LIN {X 0,Y 261.117,Z 932.425,A -85,B 0,C 180,E1 -18091.542,E2 -18091.542} C_VEL
LIN {X 0,Y 261.103,Z 931.632,A -85,B 0,C 180,E1 -18093.086,E2 -18093.086} C_VEL
LIN {X 0,Y 261.207,Z 929.523,A -85,B 0,C 180,E1 -18095.429,E2 -18095.429} C_VEL
LIN {X 0,Y 261.577,Z 926.266,A -85,B 0,C 180,E1 -18097.72,E2 -18097.72} C_VEL
LIN {X 0,Y 262.252,Z 921.503,A -85,B 0,C 180,E1 -18100.032,E2 -18100.032} C_VEL
LIN {X 0,Y 263.059,Z 916.347,A -85,B 0,C 180,E1 -18101.95,E2 -18101.95} C_VEL
LIN {X 0,Y 263.93,Z 911.311,A -85,B 0,C 180,E1 -18103.474,E2 -18103.474} C_VEL
LIN {X 0,Y 264.941,Z 905.246,A -85,B 0,C 180,E1 -18104.989,E2 -18104.989} C_VEL
LIN {X 0,Y 266.222,Z 897.871,A -85,B 0,C 180,E1 -18106.487,E2 -18106.487} C_VEL
LIN {X 0,Y 267.5,Z 889.973,A -85,B 0,C 180,E1 -18107.784,E2 -18107.784} C_VEL
LIN {X 0,Y 268.675,Z 881.626,A -85,B 0,C 180,E1 -18108.887,E2 -18108.887} C_VEL
LIN {X 0,Y 269.816,Z 871.375,A -85,B 0,C 180,E1 -18109.95,E2 -18109.95} C_VEL
LIN {X 0,Y 270.872,Z 860.075,A -85,B 0,C 180,E1 -18110.756,E2 -18110.756} C_VEL
LIN {X 0,Y 271.49,Z 850.412,A -85,B 0,C 180,E1 -18111.215,E2 -18111.215} C_VEL
LIN {X 0,Y 272.419,Z 812.541,A -85,B 0,C 180,E1 -18112.245,E2 -18112.245} C_VEL
LIN {X 0,Y 268.762,Z 786.761,A -85,B 0,C 180,E1 -18113.292,E2 -18113.292} C_VEL
LIN {X 0,Y 266.245,Z 772.739,A -85,B 0,C 180,E1 -18113.98,E2 -18113.98} C_VEL
LIN {X 0,Y 266.206,Z 769.876,A -85,B 0,C 180,E1 -18114.987,E2 -18114.987} C_VEL
LIN {X 0,Y 264.536,Z 760.93,A -85,B 0,C 180,E1 -18118.751,E2 -18118.751} C_VEL
LIN {X 0,Y 263.188,Z 754.618,A -85,B 0,C 180,E1 -18121.579,E2 -18121.579} C_VEL
LIN {X 0,Y 263.188,Z 754.5,A -85,B 0,C 180,E1 -18125.978,E2 -18125.978} C_VEL
LIN {X 0,Y 263.115,Z 754.506,A -85,B 0,C 180,E1 -18129.871,E2 -18129.871} C_VEL
LIN {X 0,Y 263.124,Z 754.518,A -85,B 0,C 180,E1 -18133.984,E2 -18133.984} C_VEL
LIN {X 0,Y 263.144,Z 754.475,A -85,B 0,C 180,E1 -18138.402,E2 -18138.402} C_VEL
LIN {X 0,Y 263.188,Z 754.456,A -85,B 0,C 180,E1 -18142.108,E2 -18142.108} C_VEL
LIN {X 0,Y 263.184,Z 754.512,A -85,B 0,C 180,E1 -18145.891,E2 -18145.891} C_VEL
LIN {X 0,Y 263.141,Z 754.502,A -85,B 0,C 180,E1 -18149.506,E2 -18149.506} C_VEL
LIN {X 0,Y 263.193,Z 754.509,A -85,B 0,C 180,E1 -18153.003,E2 -18153.003} C_VEL
LIN {X 0,Y 263.186,Z 754.503,A -85,B 0,C 180,E1 -18156.387,E2 -18156.387} C_VEL
LIN {X 0,Y 263.265,Z 754.482,A -85,B 0,C 180,E1 -18159.694,E2 -18159.694} C_VEL
LIN {X 0,Y 263.352,Z 754.487,A -85,B 0,C 180,E1 -18164.522,E2 -18164.522} C_VEL
LIN {X 0,Y 263.375,Z 754.47,A -85,B 0,C 180,E1 -18169.235,E2 -18169.235} C_VEL
LIN {X 0,Y 263.566,Z 754.468,A -85,B 0,C 180,E1 -18172.338,E2 -18172.338} C_VEL
LIN {X 0,Y 263.753,Z 754.411,A -85,B 0,C 180,E1 -18178.473,E2 -18178.473} C_VEL
LIN {X 0,Y 263.756,Z 754.439,A -85,B 0,C 180,E1 -18181.527,E2 -18181.527} C_VEL
LIN {X 0,Y 263.574,Z 754.43,A -85,B 0,C 180,E1 -18187.662,E2 -18187.662} C_VEL
LIN {X 0,Y 263.375,Z 754.483,A -85,B 0,C 180,E1 -18190.766,E2 -18190.766} C_VEL
LIN {X 0,Y 263.316,Z 754.481,A -85,B 0,C 180,E1 -18195.48,E2 -18195.48} C_VEL
LIN {X 0,Y 263.245,Z 754.501,A -85,B 0,C 180,E1 -18200.308,E2 -18200.308} C_VEL
LIN {X 0,Y 263.193,Z 754.488,A -85,B 0,C 180,E1 -18205.293,E2 -18205.293} C_VEL
LIN {X 0,Y 263.167,Z 754.512,A -85,B 0,C 180,E1 -18208.731,E2 -18208.731} C_VEL
LIN {X 0,Y 263.134,Z 754.508,A -85,B 0,C 180,E1 -18212.288,E2 -18212.288} C_VEL
LIN {X 0,Y 263.193,Z 754.513,A -85,B 0,C 180,E1 -18216.766,E2 -18216.766} C_VEL
LIN {X 0,Y 263.125,Z 754.464,A -85,B 0,C 180,E1 -18221.593,E2 -18221.593} C_VEL
LIN {X 0,Y 263.125,Z 754.512,A -85,B 0,C 180,E1 -18226.151,E2 -18226.151} C_VEL
LIN {X 0,Y 263.107,Z 754.502,A -85,B 0,C 180,E1 -18230.128,E2 -18230.128} C_VEL
LIN {X 0,Y 263.164,Z 754.51,A -85,B 0,C 180,E1 -18234.018,E2 -18234.018} C_VEL
LIN {X 0,Y 263.129,Z 754.501,A -85,B 0,C 180,E1 -18237.711,E2 -18237.711} C_VEL
LIN {X 0,Y 263.149,Z 754.515,A -85,B 0,C 180,E1 -18241.805,E2 -18241.805} C_VEL
LIN {X 0,Y 263.218,Z 754.632,A -85,B 0,C 180,E1 -18243.861,E2 -18243.861} C_VEL
LIN {X 0,Y 264.092,Z 758.93,A -85,B 0,C 180,E1 -18245.847,E2 -18245.847} C_VEL
LIN {X 0,Y 265.718,Z 763.312,A -85,B 0,C 180,E1 -18246.209,E2 -18246.209} C_VEL
LIN {X 0,Y 270.426,Z 776.032,A -85,B 0,C 180,E1 -18247.014,E2 -18247.014} C_VEL
LIN {X 0,Y 272.953,Z 789.739,A -85,B 0,C 180,E1 -18247.624,E2 -18247.624} C_VEL
LIN {X 0,Y 271.82,Z 834.743,A -85,B 0,C 180,E1 -18248.828,E2 -18248.828} C_VEL
LIN {X 0,Y 271.425,Z 844.466,A -85,B 0,C 180,E1 -18249.292,E2 -18249.292} C_VEL
LIN {X 0,Y 270.462,Z 855.519,A -85,B 0,C 180,E1 -18250.059,E2 -18250.059} C_VEL
LIN {X 0,Y 269.384,Z 866.303,A -85,B 0,C 180,E1 -18251.164,E2 -18251.164} C_VEL
LIN {X 0,Y 268.158,Z 874.683,A -85,B 0,C 180,E1 -18252.261,E2 -18252.261} C_VEL
LIN {X 0,Y 267.02,Z 882.591,A -85,B 0,C 180,E1 -18253.564,E2 -18253.564} C_VEL
LIN {X 0,Y 266.157,Z 888.266,A -85,B 0,C 180,E1 -18254.689,E2 -18254.689} C_VEL
LIN {X 0,Y 265.023,Z 894.607,A -85,B 0,C 180,E1 -18256.192,E2 -18256.192} C_VEL
LIN {X 0,Y 264.038,Z 899.876,A -85,B 0,C 180,E1 -18257.705,E2 -18257.705} C_VEL
LIN {X 0,Y 263.243,Z 904.272,A -85,B 0,C 180,E1 -18259.229,E2 -18259.229} C_VEL
LIN {X 0,Y 262.4,Z 909.439,A -85,B 0,C 180,E1 -18261.529,E2 -18261.529} C_VEL
LIN {X 0,Y 261.9,Z 912.232,A -85,B 0,C 180,E1 -18263.161,E2 -18263.161} C_VEL
LIN {X 0,Y 261.498,Z 914.99,A -85,B 0,C 180,E1 -18265.375,E2 -18265.375} C_VEL
LIN {X 0,Y 261.304,Z 916.256,A -85,B 0,C 180,E1 -18266.916,E2 -18266.916} C_VEL
LIN {X 0,Y 261.17,Z 917.054,A -85,B 0,C 180,E1 -18268.458,E2 -18268.458} C_VEL
LIN {X 0,Y 261.135,Z 917.357,A -85,B 0,C 180,E1 -18270,E2 -18270} C_VEL
LIN {X 0,Y 261.168,Z 917.078,A -85,B 0,C 180,E1 -18271.542,E2 -18271.542} C_VEL
LIN {X 0,Y 261.298,Z 916.33,A -85,B 0,C 180,E1 -18273.084,E2 -18273.084} C_VEL
LIN {X 0,Y 261.492,Z 915.114,A -85,B 0,C 180,E1 -18274.625,E2 -18274.625} C_VEL
LIN {X 0,Y 261.9,Z 912.408,A -85,B 0,C 180,E1 -18276.839,E2 -18276.839} C_VEL
LIN {X 0,Y 262.343,Z 909.671,A -85,B 0,C 180,E1 -18278.473,E2 -18278.473} C_VEL
LIN {X 0,Y 263.189,Z 904.567,A -85,B 0,C 180,E1 -18280.773,E2 -18280.773} C_VEL
LIN {X 0,Y 264.251,Z 899.069,A -85,B 0,C 180,E1 -18282.675,E2 -18282.675} C_VEL
LIN {X 0,Y 265.54,Z 892.157,A -85,B 0,C 180,E1 -18284.562,E2 -18284.562} C_VEL
LIN {X 0,Y 266.805,Z 884.221,A -85,B 0,C 180,E1 -18286.253,E2 -18286.253} C_VEL
LIN {X 0,Y 267.939,Z 876.65,A -85,B 0,C 180,E1 -18287.556,E2 -18287.556} C_VEL
LIN {X 0,Y 269.095,Z 868.708,A -85,B 0,C 180,E1 -18288.659,E2 -18288.659} C_VEL
LIN {X 0,Y 270.084,Z 860.5,A -85,B 0,C 180,E1 -18289.574,E2 -18289.574} C_VEL
LIN {X 0,Y 270.945,Z 852.17,A -85,B 0,C 180,E1 -18290.3,E2 -18290.3} C_VEL
LIN {X 0,Y 271.513,Z 843.152,A -85,B 0,C 180,E1 -18290.899,E2 -18290.899} C_VEL
LIN {X 0,Y 271.912,Z 833.656,A -85,B 0,C 180,E1 -18291.326,E2 -18291.326} C_VEL
LIN {X 0,Y 272.955,Z 789.105,A -85,B 0,C 180,E1 -18292.514,E2 -18292.514} C_VEL
LIN {X 0,Y 270.294,Z 775.622,A -85,B 0,C 180,E1 -18293.131,E2 -18293.131} C_VEL
LIN {X 0,Y 265.133,Z 761.667,A -85,B 0,C 180,E1 -18294.018,E2 -18294.018} C_VEL
LIN {X 0,Y 264.195,Z 759.242,A -85,B 0,C 180,E1 -18294.218,E2 -18294.218} C_VEL
LIN {X 0,Y 264.031,Z 758.561,A -85,B 0,C 180,E1 -18294.368,E2 -18294.368} C_VEL
LIN {X 0,Y 263.208,Z 754.591,A -85,B 0,C 180,E1 -18296.354,E2 -18296.354} C_VEL
LIN {X 0,Y 263.127,Z 754.51,A -85,B 0,C 180,E1 -18300.496,E2 -18300.496} C_VEL
LIN {X 0,Y 263.152,Z 754.518,A -85,B 0,C 180,E1 -18304.114,E2 -18304.114} C_VEL
LIN {X 0,Y 263.16,Z 754.486,A -85,B 0,C 180,E1 -18307.897,E2 -18307.897} C_VEL
LIN {X 0,Y 263.125,Z 754.52,A -85,B 0,C 180,E1 -18311.893,E2 -18311.893} C_VEL
LIN {X 0,Y 263.106,Z 754.474,A -85,B 0,C 180,E1 -18316.155,E2 -18316.155} C_VEL
LIN {X 0,Y 263.106,Z 754.494,A -85,B 0,C 180,E1 -18320.127,E2 -18320.127} C_VEL
LIN {X 0,Y 263.176,Z 754.514,A -85,B 0,C 180,E1 -18324.02,E2 -18324.02} C_VEL
LIN {X 0,Y 263.134,Z 754.506,A -85,B 0,C 180,E1 -18327.712,E2 -18327.712} C_VEL
LIN {X 0,Y 263.197,Z 754.507,A -85,B 0,C 180,E1 -18331.785,E2 -18331.785} C_VEL
LIN {X 0,Y 263.202,Z 754.49,A -85,B 0,C 180,E1 -18335.212,E2 -18335.212} C_VEL
LIN {X 0,Y 263.263,Z 754.499,A -85,B 0,C 180,E1 -18339.693,E2 -18339.693} C_VEL
LIN {X 0,Y 263.316,Z 754.481,A -85,B 0,C 180,E1 -18344.52,E2 -18344.52} C_VEL
LIN {X 0,Y 263.375,Z 754.484,A -85,B 0,C 180,E1 -18349.234,E2 -18349.234} C_VEL
LIN {X 0,Y 263.574,Z 754.43,A -85,B 0,C 180,E1 -18352.338,E2 -18352.338} C_VEL
LIN {X 0,Y 263.756,Z 754.439,A -85,B 0,C 180,E1 -18358.473,E2 -18358.473} C_VEL
LIN {X 0,Y 263.752,Z 754.411,A -85,B 0,C 180,E1 -18361.527,E2 -18361.527} C_VEL
LIN {X 0,Y 263.58,Z 754.43,A -85,B 0,C 180,E1 -18362.831,E2 -18362.831} C_VEL
LIN {X 0,Y 262.872,Z 754.533,A -85,B 0,C 180,E1 -18364.106,E2 -18364.106} C_VEL
LIN {X 0,Y 260.07,Z 754.901,A -85,B 0,C 180,E1 -18366.185,E2 -18366.185} C_VEL
LIN {X 0,Y 256.828,Z 755.305,A -85,B 0,C 180,E1 -18368.741,E2 -18368.741} C_VEL
LIN {X 0,Y 256.429,Z 755.343,A -85,B 0,C 180,E1 -18369.626,E2 -18369.626} C_VEL
LIN {X 0,Y 256.257,Z 755.361,A -85,B 0,C 180,E1 -18374.29,E2 -18374.29} C_VEL
LIN {X 0,Y 256.213,Z 755.383,A -85,B 0,C 180,E1 -18377.562,E2 -18377.562} C_VEL
LIN {X 0,Y 256.159,Z 755.361,A -85,B 0,C 180,E1 -18381.12,E2 -18381.12} C_VEL
LIN {X 0,Y 256.189,Z 755.384,A -85,B 0,C 180,E1 -18385.138,E2 -18385.138} C_VEL
LIN {X 0,Y 256.104,Z 755.373,A -85,B 0,C 180,E1 -18389.601,E2 -18389.601} C_VEL
LIN {X 0,Y 256.086,Z 755.398,A -85,B 0,C 180,E1 -18393.29,E2 -18393.29} C_VEL
LIN {X 0,Y 256.14,Z 755.342,A -85,B 0,C 180,E1 -18397.278,E2 -18397.278} C_VEL
LIN {X 0,Y 256.076,Z 755.348,A -85,B 0,C 180,E1 -18401.199,E2 -18401.199} C_VEL
LIN {X 0,Y 256.06,Z 755.4,A -85,B 0,C 180,E1 -18405.53,E2 -18405.53} C_VEL
LIN {X 0,Y 256.056,Z 755.373,A -85,B 0,C 180,E1 -18408.797,E2 -18408.797} C_VEL
LIN {X 0,Y 256.145,Z 755.383,A -85,B 0,C 180,E1 -18412.87,E2 -18412.87} C_VEL
LIN {X 0,Y 256.094,Z 755.392,A -85,B 0,C 180,E1 -18416.711,E2 -18416.711} C_VEL
LIN {X 0,Y 256.157,Z 755.646,A -85,B 0,C 180,E1 -18418,E2 -18418} C_VEL
LIN {X 0,Y 257.849,Z 763.676,A -85,B 0,C 180,E1 -18421.651,E2 -18421.651} C_VEL
LIN {X 0,Y 259.382,Z 772.257,A -85,B 0,C 180,E1 -18425.261,E2 -18425.261} C_VEL
LIN {X 0,Y 259.914,Z 775.065,A -85,B 0,C 180,E1 -18425.493,E2 -18425.493} C_VEL
LIN {X 0,Y 263.741,Z 797.233,A -85,B 0,C 180,E1 -18426.514,E2 -18426.514} C_VEL
LIN {X 0,Y 265.925,Z 814.859,A -85,B 0,C 180,E1 -18427.222,E2 -18427.222} C_VEL
LIN {X 0,Y 264.928,Z 850.11,A -85,B 0,C 180,E1 -18428.199,E2 -18428.199} C_VEL
LIN {X 0,Y 264.155,Z 861.586,A -85,B 0,C 180,E1 -18428.767,E2 -18428.767} C_VEL
LIN {X 0,Y 263.016,Z 872.951,A -85,B 0,C 180,E1 -18429.673,E2 -18429.673} C_VEL
LIN {X 0,Y 261.922,Z 881.642,A -85,B 0,C 180,E1 -18430.607,E2 -18430.607} C_VEL
LIN {X 0,Y 260.751,Z 889.947,A -85,B 0,C 180,E1 -18431.74,E2 -18431.74} C_VEL
LIN {X 0,Y 259.427,Z 897.809,A -85,B 0,C 180,E1 -18433.069,E2 -18433.069} C_VEL
LIN {X 0,Y 258.085,Z 905.162,A -85,B 0,C 180,E1 -18434.603,E2 -18434.603} C_VEL
LIN {X 0,Y 256.786,Z 912.628,A -85,B 0,C 180,E1 -18436.548,E2 -18436.548} C_VEL
LIN {X 0,Y 255.534,Z 919.443,A -85,B 0,C 180,E1 -18438.9,E2 -18438.9} C_VEL
LIN {X 0,Y 254.702,Z 924.626,A -85,B 0,C 180,E1 -18441.271,E2 -18441.271} C_VEL
LIN {X 0,Y 254.238,Z 928.436,A -85,B 0,C 180,E1 -18443.652,E2 -18443.652} C_VEL
LIN {X 0,Y 254.061,Z 930.186,A -85,B 0,C 180,E1 -18445.24,E2 -18445.24} C_VEL
LIN {X 0,Y 254.003,Z 931.441,A -85,B 0,C 180,E1 -18446.828,E2 -18446.828} C_VEL
LIN {X 0,Y 254.024,Z 932.222,A -85,B 0,C 180,E1 -18448.415,E2 -18448.415} C_VEL
LIN {X 0,Y 254.054,Z 932.517,A -85,B 0,C 180,E1 -18450,E2 -18450} C_VEL
LIN {X 0,Y 254.024,Z 932.216,A -85,B 0,C 180,E1 -18451.585,E2 -18451.585} C_VEL
LIN {X 0,Y 254.003,Z 931.423,A -85,B 0,C 180,E1 -18453.172,E2 -18453.172} C_VEL
LIN {X 0,Y 254.093,Z 929.602,A -85,B 0,C 180,E1 -18455.299,E2 -18455.299} C_VEL
LIN {X 0,Y 254.525,Z 926.055,A -85,B 0,C 180,E1 -18457.936,E2 -18457.936} C_VEL
LIN {X 0,Y 255.234,Z 921.292,A -85,B 0,C 180,E1 -18460.31,E2 -18460.31} C_VEL
LIN {X 0,Y 256.088,Z 916.135,A -85,B 0,C 180,E1 -18462.28,E2 -18462.28} C_VEL
LIN {X 0,Y 257.013,Z 911.099,A -85,B 0,C 180,E1 -18463.843,E2 -18463.843} C_VEL
LIN {X 0,Y 258.08,Z 905.034,A -85,B 0,C 180,E1 -18465.397,E2 -18465.397} C_VEL
LIN {X 0,Y 259.406,Z 897.658,A -85,B 0,C 180,E1 -18466.933,E2 -18466.933} C_VEL
LIN {X 0,Y 260.745,Z 889.761,A -85,B 0,C 180,E1 -18468.26,E2 -18468.26} C_VEL
LIN {X 0,Y 261.949,Z 881.412,A -85,B 0,C 180,E1 -18469.391,E2 -18469.391} C_VEL
LIN {X 0,Y 263.121,Z 871.423,A -85,B 0,C 180,E1 -18470.453,E2 -18470.453} C_VEL
LIN {X 0,Y 264.277,Z 859.339,A -85,B 0,C 180,E1 -18471.331,E2 -18471.331} C_VEL
LIN {X 0,Y 264.881,Z 850.416,A -85,B 0,C 180,E1 -18471.762,E2 -18471.762} C_VEL
LIN {X 0,Y 265.597,Z 821.575,A -85,B 0,C 180,E1 -18472.583,E2 -18472.583} C_VEL
LIN {X 0,Y 265.746,Z 812.432,A -85,B 0,C 180,E1 -18472.831,E2 -18472.831} C_VEL
LIN {X 0,Y 261.818,Z 785.322,A -85,B 0,C 180,E1 -18473.983,E2 -18473.983} C_VEL
LIN {X 0,Y 259.445,Z 772.931,A -85,B 0,C 180,E1 -18474.608,E2 -18474.608} C_VEL
LIN {X 0,Y 259.328,Z 771.853,A -85,B 0,C 180,E1 -18474.838,E2 -18474.838} C_VEL
LIN {X 0,Y 257.819,Z 763.609,A -85,B 0,C 180,E1 -18478.352,E2 -18478.352} C_VEL
LIN {X 0,Y 256.158,Z 755.594,A -85,B 0,C 180,E1 -18482.001,E2 -18482.001} C_VEL
LIN {X 0,Y 256.121,Z 755.382,A -85,B 0,C 180,E1 -18485.187,E2 -18485.187} C_VEL
LIN {X 0,Y 256.088,Z 755.391,A -85,B 0,C 180,E1 -18489.139,E2 -18489.139} C_VEL
LIN {X 0,Y 256.062,Z 755.39,A -85,B 0,C 180,E1 -18493.327,E2 -18493.327} C_VEL
LIN {X 0,Y 256.086,Z 755.367,A -85,B 0,C 180,E1 -18497.816,E2 -18497.816} C_VEL
LIN {X 0,Y 256.1,Z 755.327,A -85,B 0,C 180,E1 -18500.863,E2 -18500.863} C_VEL
LIN {X 0,Y 256.122,Z 755.385,A -85,B 0,C 180,E1 -18504.814,E2 -18504.814} C_VEL
LIN {X 0,Y 256.093,Z 755.39,A -85,B 0,C 180,E1 -18508.573,E2 -18508.573} C_VEL
LIN {X 0,Y 256.139,Z 755.38,A -85,B 0,C 180,E1 -18512.196,E2 -18512.196} C_VEL
LIN {X 0,Y 256.168,Z 755.384,A -85,B 0,C 180,E1 -18515.699,E2 -18515.699} C_VEL
LIN {X 0,Y 256.168,Z 755.361,A -85,B 0,C 180,E1 -18519.105,E2 -18519.105} C_VEL
LIN {X 0,Y 256.301,Z 755.369,A -85,B 0,C 180,E1 -18524.085,E2 -18524.085} C_VEL
LIN {X 0,Y 256.311,Z 755.345,A -85,B 0,C 180,E1 -18528.934,E2 -18528.934} C_VEL
LIN {X 0,Y 256.529,Z 755.342,A -85,B 0,C 180,E1 -18532.127,E2 -18532.127} C_VEL
LIN {X 0,Y 256.5,Z 755.313,A -85,B 0,C 180,E1 -18536.859,E2 -18536.859} C_VEL
LIN {X 0,Y 256.768,Z 755.298,A -85,B 0,C 180,E1 -18540,E2 -18540} C_VEL
LIN {X 0,Y 256.507,Z 755.343,A -85,B 0,C 180,E1 -18543.141,E2 -18543.141} C_VEL
LIN {X 0,Y 256.542,Z 755.306,A -85,B 0,C 180,E1 -18547.873,E2 -18547.873} C_VEL
LIN {X 0,Y 256.311,Z 755.366,A -85,B 0,C 180,E1 -18551.066,E2 -18551.066} C_VEL
LIN {X 0,Y 256.238,Z 755.374,A -85,B 0,C 180,E1 -18554.291,E2 -18554.291} C_VEL
LIN {X 0,Y 256.182,Z 755.357,A -85,B 0,C 180,E1 -18557.564,E2 -18557.564} C_VEL
LIN {X 0,Y 256.144,Z 755.392,A -85,B 0,C 180,E1 -18561.111,E2 -18561.111} C_VEL
LIN {X 0,Y 256.172,Z 755.363,A -85,B 0,C 180,E1 -18565.13,E2 -18565.13} C_VEL
LIN {X 0,Y 256.105,Z 755.396,A -85,B 0,C 180,E1 -18569.601,E2 -18569.601} C_VEL
LIN {X 0,Y 256.069,Z 755.381,A -85,B 0,C 180,E1 -18573.293,E2 -18573.293} C_VEL
LIN {X 0,Y 256.122,Z 755.394,A -85,B 0,C 180,E1 -18577.273,E2 -18577.273} C_VEL
LIN {X 0,Y 256.055,Z 755.348,A -85,B 0,C 180,E1 -18581.204,E2 -18581.204} C_VEL
LIN {X 0,Y 256.055,Z 755.384,A -85,B 0,C 180,E1 -18585.531,E2 -18585.531} C_VEL
LIN {X 0,Y 256.056,Z 755.398,A -85,B 0,C 180,E1 -18588.797,E2 -18588.797} C_VEL
LIN {X 0,Y 256.131,Z 755.366,A -85,B 0,C 180,E1 -18592.867,E2 -18592.867} C_VEL
LIN {X 0,Y 256.067,Z 755.391,A -85,B 0,C 180,E1 -18596.707,E2 -18596.707} C_VEL
LIN {X 0,Y 256.056,Z 755.401,A -85,B 0,C 180,E1 -18600.393,E2 -18600.393} C_VEL
LIN {X 0,Y 256.17,Z 755.527,A -85,B 0,C 180,E1 -18603.414,E2 -18603.414} C_VEL
LIN {X 0,Y 256.885,Z 758.981,A -85,B 0,C 180,E1 -18605.088,E2 -18605.088} C_VEL
LIN {X 0,Y 257.529,Z 760.941,A -85,B 0,C 180,E1 -18605.323,E2 -18605.323} C_VEL
LIN {X 0,Y 263.776,Z 777.152,A -85,B 0,C 180,E1 -18606.425,E2 -18606.425} C_VEL
LIN {X 0,Y 266.333,Z 789.717,A -85,B 0,C 180,E1 -18607.029,E2 -18607.029} C_VEL
LIN {X 0,Y 265.234,Z 834.968,A -85,B 0,C 180,E1 -18608.276,E2 -18608.276} C_VEL
LIN {X 0,Y 264.81,Z 844.686,A -85,B 0,C 180,E1 -18608.75,E2 -18608.75} C_VEL
LIN {X 0,Y 263.821,Z 855.735,A -85,B 0,C 180,E1 -18609.535,E2 -18609.535} C_VEL
LIN {X 0,Y 262.675,Z 866.517,A -85,B 0,C 180,E1 -18610.664,E2 -18610.664} C_VEL
LIN {X 0,Y 261.427,Z 874.896,A -85,B 0,C 180,E1 -18611.789,E2 -18611.789} C_VEL
LIN {X 0,Y 260.236,Z 882.802,A -85,B 0,C 180,E1 -18613.123,E2 -18613.123} C_VEL
LIN {X 0,Y 259.329,Z 888.477,A -85,B 0,C 180,E1 -18614.276,E2 -18614.276} C_VEL
LIN {X 0,Y 258.126,Z 894.818,A -85,B 0,C 180,E1 -18615.816,E2 -18615.816} C_VEL
LIN {X 0,Y 257.122,Z 900.086,A -85,B 0,C 180,E1 -18617.369,E2 -18617.369} C_VEL
LIN {X 0,Y 256.29,Z 904.482,A -85,B 0,C 180,E1 -18618.933,E2 -18618.933} C_VEL
LIN {X 0,Y 255.386,Z 909.649,A -85,B 0,C 180,E1 -18621.295,E2 -18621.295} C_VEL
LIN {X 0,Y 254.785,Z 912.819,A -85,B 0,C 180,E1 -18623.231,E2 -18623.231} C_VEL
LIN {X 0,Y 254.435,Z 915.199,A -85,B 0,C 180,E1 -18625.247,E2 -18625.247} C_VEL
LIN {X 0,Y 254.223,Z 916.465,A -85,B 0,C 180,E1 -18626.83,E2 -18626.83} C_VEL
LIN {X 0,Y 254.102,Z 917.262,A -85,B 0,C 180,E1 -18628.415,E2 -18628.415} C_VEL
LIN {X 0,Y 254.063,Z 917.565,A -85,B 0,C 180,E1 -18630,E2 -18630} C_VEL
LIN {X 0,Y 254.099,Z 917.286,A -85,B 0,C 180,E1 -18631.585,E2 -18631.585} C_VEL
LIN {X 0,Y 254.218,Z 916.538,A -85,B 0,C 180,E1 -18633.17,E2 -18633.17} C_VEL
LIN {X 0,Y 254.429,Z 915.322,A -85,B 0,C 180,E1 -18634.753,E2 -18634.753} C_VEL
LIN {X 0,Y 254.775,Z 913.02,A -85,B 0,C 180,E1 -18636.751,E2 -18636.751} C_VEL
LIN {X 0,Y 255.314,Z 909.879,A -85,B 0,C 180,E1 -18638.708,E2 -18638.708} C_VEL
LIN {X 0,Y 256.212,Z 904.774,A -85,B 0,C 180,E1 -18641.07,E2 -18641.07} C_VEL
LIN {X 0,Y 257.322,Z 899.276,A -85,B 0,C 180,E1 -18643.022,E2 -18643.022} C_VEL
LIN {X 0,Y 258.682,Z 892.363,A -85,B 0,C 180,E1 -18644.957,E2 -18644.957} C_VEL
LIN {X 0,Y 259.972,Z 884.427,A -85,B 0,C 180,E1 -18646.692,E2 -18646.692} C_VEL
LIN {X 0,Y 261.176,Z 876.855,A -85,B 0,C 180,E1 -18648.026,E2 -18648.026} C_VEL
LIN {X 0,Y 262.402,Z 868.912,A -85,B 0,C 180,E1 -18649.153,E2 -18649.153} C_VEL
LIN {X 0,Y 263.412,Z 860.702,A -85,B 0,C 180,E1 -18650.091,E2 -18650.091} C_VEL
LIN {X 0,Y 264.313,Z 852.37,A -85,B 0,C 180,E1 -18650.833,E2 -18650.833} C_VEL
LIN {X 0,Y 264.909,Z 843.349,A -85,B 0,C 180,E1 -18651.445,E2 -18651.445} C_VEL
LIN {X 0,Y 265.325,Z 834.442,A -85,B 0,C 180,E1 -18651.859,E2 -18651.859} C_VEL
LIN {X 0,Y 266.399,Z 789.956,A -85,B 0,C 180,E1 -18653.08,E2 -18653.08} C_VEL
LIN {X 0,Y 263.941,Z 777.61,A -85,B 0,C 180,E1 -18653.669,E2 -18653.669} C_VEL
LIN {X 0,Y 258.029,Z 762.029,A -85,B 0,C 180,E1 -18654.718,E2 -18654.718} C_VEL
LIN {X 0,Y 256.954,Z 759.158,A -85,B 0,C 180,E1 -18654.996,E2 -18654.996} C_VEL
LIN {X 0,Y 256.165,Z 755.549,A -85,B 0,C 180,E1 -18656.696,E2 -18656.696} C_VEL
LIN {X 0,Y 256.083,Z 755.378,A -85,B 0,C 180,E1 -18661.429,E2 -18661.429} C_VEL
LIN {X 0,Y 256.083,Z 755.403,A -85,B 0,C 180,E1 -18665.193,E2 -18665.193} C_VEL
LIN {X 0,Y 256.115,Z 755.368,A -85,B 0,C 180,E1 -18667.27,E2 -18667.27} C_VEL
LIN {X 0,Y 256.056,Z 755.395,A -85,B 0,C 180,E1 -18671.203,E2 -18671.203} C_VEL
LIN {X 0,Y 256.045,Z 755.363,A -85,B 0,C 180,E1 -18675.533,E2 -18675.533} C_VEL
LIN {X 0,Y 256.055,Z 755.347,A -85,B 0,C 180,E1 -18678.796,E2 -18678.796} C_VEL
LIN {X 0,Y 256.138,Z 755.393,A -85,B 0,C 180,E1 -18682.869,E2 -18682.869} C_VEL
LIN {X 0,Y 256.069,Z 755.381,A -85,B 0,C 180,E1 -18686.707,E2 -18686.707} C_VEL
LIN {X 0,Y 256.105,Z 755.396,A -85,B 0,C 180,E1 -18690.399,E2 -18690.399} C_VEL
LIN {X 0,Y 256.172,Z 755.363,A -85,B 0,C 180,E1 -18694.87,E2 -18694.87} C_VEL
LIN {X 0,Y 256.164,Z 755.388,A -85,B 0,C 180,E1 -18699.104,E2 -18699.104} C_VEL
LIN {X 0,Y 256.235,Z 755.354,A -85,B 0,C 180,E1 -18703.735,E2 -18703.735} C_VEL
LIN {X 0,Y 256.292,Z 755.375,A -85,B 0,C 180,E1 -18707.327,E2 -18707.327} C_VEL
LIN {X 0,Y 256.498,Z 755.328,A -85,B 0,C 180,E1 -18710.538,E2 -18710.538} C_VEL
LIN {X 0,Y 256.489,Z 755.32,A -85,B 0,C 180,E1 -18713.707,E2 -18713.707} C_VEL
LIN {X 0,Y 256.719,Z 755.315,A -85,B 0,C 180,E1 -18718.431,E2 -18718.431} C_VEL
LIN {X 0,Y 256.715,Z 755.287,A -85,B 0,C 180,E1 -18721.569,E2 -18721.569} C_VEL
LIN {X 0,Y 256.484,Z 755.347,A -85,B 0,C 180,E1 -18726.292,E2 -18726.292} C_VEL
LIN {X 0,Y 256.429,Z 755.343,A -85,B 0,C 180,E1 -18729.626,E2 -18729.626} C_VEL
LIN {X 0,Y 255.655,Z 755.431,A -85,B 0,C 180,E1 -18730.934,E2 -18730.934} C_VEL
LIN {X 0,Y 252.801,Z 755.795,A -85,B 0,C 180,E1 -18733.068,E2 -18733.068} C_VEL
LIN {X 0,Y 249.582,Z 756.211,A -85,B 0,C 180,E1 -18735.695,E2 -18735.695} C_VEL
LIN {X 0,Y 249.208,Z 756.253,A -85,B 0,C 180,E1 -18736.604,E2 -18736.604} C_VEL
LIN {X 0,Y 249.089,Z 756.241,A -85,B 0,C 180,E1 -18741.518,E2 -18741.518} C_VEL
LIN {X 0,Y 249.131,Z 756.264,A -85,B 0,C 180,E1 -18745.482,E2 -18745.482} C_VEL
LIN {X 0,Y 249.074,Z 756.249,A -85,B 0,C 180,E1 -18748.989,E2 -18748.989} C_VEL
LIN {X 0,Y 249.037,Z 756.277,A -85,B 0,C 180,E1 -18752.425,E2 -18752.425} C_VEL
LIN {X 0,Y 249.075,Z 756.242,A -85,B 0,C 180,E1 -18756.338,E2 -18756.338} C_VEL
LIN {X 0,Y 249.035,Z 756.212,A -85,B 0,C 180,E1 -18760.472,E2 -18760.472} C_VEL
LIN {X 0,Y 249.006,Z 756.281,A -85,B 0,C 180,E1 -18764.878,E2 -18764.878} C_VEL
LIN {X 0,Y 249.017,Z 756.256,A -85,B 0,C 180,E1 -18767.363,E2 -18767.363} C_VEL
LIN {X 0,Y 249.038,Z 756.277,A -85,B 0,C 180,E1 -18771.622,E2 -18771.622} C_VEL
LIN {X 0,Y 249.063,Z 756.268,A -85,B 0,C 180,E1 -18775.642,E2 -18775.642} C_VEL
LIN {X 0,Y 249.102,Z 756.505,A -85,B 0,C 180,E1 -18777.465,E2 -18777.465} C_VEL
LIN {X 0,Y 250.689,Z 764.037,A -85,B 0,C 180,E1 -18781.011,E2 -18781.011} C_VEL
LIN {X 0,Y 252.179,Z 771.969,A -85,B 0,C 180,E1 -18784.49,E2 -18784.49} C_VEL
LIN {X 0,Y 253.032,Z 774.773,A -85,B 0,C 180,E1 -18784.778,E2 -18784.778} C_VEL
LIN {X 0,Y 256.168,Z 791.111,A -85,B 0,C 180,E1 -18785.598,E2 -18785.598} C_VEL
LIN {X 0,Y 259.352,Z 814.102,A -85,B 0,C 180,E1 -18786.594,E2 -18786.594} C_VEL
LIN {X 0,Y 258.366,Z 849.917,A -85,B 0,C 180,E1 -18787.615,E2 -18787.615} C_VEL
LIN {X 0,Y 257.558,Z 861.341,A -85,B 0,C 180,E1 -18788.192,E2 -18788.192} C_VEL
LIN {X 0,Y 256.374,Z 872.748,A -85,B 0,C 180,E1 -18789.123,E2 -18789.123} C_VEL
LIN {X 0,Y 255.236,Z 881.437,A -85,B 0,C 180,E1 -18790.077,E2 -18790.077} C_VEL
LIN {X 0,Y 254.008,Z 889.741,A -85,B 0,C 180,E1 -18791.237,E2 -18791.237} C_VEL
LIN {X 0,Y 252.638,Z 897.603,A -85,B 0,C 180,E1 -18792.6,E2 -18792.6} C_VEL
LIN {X 0,Y 251.247,Z 904.956,A -85,B 0,C 180,E1 -18794.173,E2 -18794.173} C_VEL
LIN {X 0,Y 249.866,Z 912.42,A -85,B 0,C 180,E1 -18796.168,E2 -18796.168} C_VEL
LIN {X 0,Y 248.56,Z 919.236,A -85,B 0,C 180,E1 -18798.584,E2 -18798.584} C_VEL
LIN {X 0,Y 247.677,Z 924.418,A -85,B 0,C 180,E1 -18801.021,E2 -18801.021} C_VEL
LIN {X 0,Y 247.176,Z 928.227,A -85,B 0,C 180,E1 -18803.469,E2 -18803.469} C_VEL
LIN {X 0,Y 246.969,Z 929.978,A -85,B 0,C 180,E1 -18805.103,E2 -18805.103} C_VEL
LIN {X 0,Y 246.907,Z 931.232,A -85,B 0,C 180,E1 -18806.736,E2 -18806.736} C_VEL
LIN {X 0,Y 246.933,Z 932.014,A -85,B 0,C 180,E1 -18808.369,E2 -18808.369} C_VEL
LIN {X 0,Y 246.983,Z 932.309,A -85,B 0,C 180,E1 -18810,E2 -18810} C_VEL
LIN {X 0,Y 246.933,Z 932.007,A -85,B 0,C 180,E1 -18811.631,E2 -18811.631} C_VEL
LIN {X 0,Y 246.907,Z 931.213,A -85,B 0,C 180,E1 -18813.264,E2 -18813.264} C_VEL
LIN {X 0,Y 246.984,Z 929.674,A -85,B 0,C 180,E1 -18815.169,E2 -18815.169} C_VEL
LIN {X 0,Y 247.301,Z 927.022,A -85,B 0,C 180,E1 -18817.347,E2 -18817.347} C_VEL
LIN {X 0,Y 247.676,Z 924.359,A -85,B 0,C 180,E1 -18818.979,E2 -18818.979} C_VEL
LIN {X 0,Y 248.553,Z 919.158,A -85,B 0,C 180,E1 -18821.416,E2 -18821.416} C_VEL
LIN {X 0,Y 249.865,Z 912.306,A -85,B 0,C 180,E1 -18823.832,E2 -18823.832} C_VEL
LIN {X 0,Y 251.241,Z 904.823,A -85,B 0,C 180,E1 -18825.827,E2 -18825.827} C_VEL
LIN {X 0,Y 252.623,Z 897.446,A -85,B 0,C 180,E1 -18827.402,E2 -18827.402} C_VEL
LIN {X 0,Y 254.002,Z 889.548,A -85,B 0,C 180,E1 -18828.763,E2 -18828.763} C_VEL
LIN {X 0,Y 255.267,Z 881.199,A -85,B 0,C 180,E1 -18829.92,E2 -18829.92} C_VEL
LIN {X 0,Y 256.595,Z 870.218,A -85,B 0,C 180,E1 -18831.099,E2 -18831.099} C_VEL
LIN {X 0,Y 257.685,Z 858.914,A -85,B 0,C 180,E1 -18831.917,E2 -18831.917} C_VEL
LIN {X 0,Y 258.367,Z 849.079,A -85,B 0,C 180,E1 -18832.385,E2 -18832.385} C_VEL
LIN {X 0,Y 259.157,Z 812.947,A -85,B 0,C 180,E1 -18833.424,E2 -18833.424} C_VEL
LIN {X 0,Y 255.401,Z 786.709,A -85,B 0,C 180,E1 -18834.576,E2 -18834.576} C_VEL
LIN {X 0,Y 252.976,Z 774.637,A -85,B 0,C 180,E1 -18835.195,E2 -18835.195} C_VEL
LIN {X 0,Y 252.242,Z 772.158,A -85,B 0,C 180,E1 -18835.427,E2 -18835.427} C_VEL
LIN {X 0,Y 250.677,Z 763.961,A -85,B 0,C 180,E1 -18838.988,E2 -18838.988} C_VEL
LIN {X 0,Y 249.093,Z 756.324,A -85,B 0,C 180,E1 -18842.656,E2 -18842.656} C_VEL
LIN {X 0,Y 249.069,Z 756.258,A -85,B 0,C 180,E1 -18846.339,E2 -18846.339} C_VEL
LIN {X 0,Y 249.026,Z 756.252,A -85,B 0,C 180,E1 -18850.474,E2 -18850.474} C_VEL
LIN {X 0,Y 249.006,Z 756.28,A -85,B 0,C 180,E1 -18854.879,E2 -18854.879} C_VEL
LIN {X 0,Y 249.027,Z 756.255,A -85,B 0,C 180,E1 -18857.365,E2 -18857.365} C_VEL
LIN {X 0,Y 249.048,Z 756.209,A -85,B 0,C 180,E1 -18861.624,E2 -18861.624} C_VEL
LIN {X 0,Y 249.062,Z 756.269,A -85,B 0,C 180,E1 -18865.643,E2 -18865.643} C_VEL
LIN {X 0,Y 249.048,Z 756.257,A -85,B 0,C 180,E1 -18869.473,E2 -18869.473} C_VEL
LIN {X 0,Y 249.073,Z 756.268,A -85,B 0,C 180,E1 -18873.162,E2 -18873.162} C_VEL
LIN {X 0,Y 249.081,Z 756.258,A -85,B 0,C 180,E1 -18876.733,E2 -18876.733} C_VEL
LIN {X 0,Y 249.112,Z 756.248,A -85,B 0,C 180,E1 -18880.212,E2 -18880.212} C_VEL
LIN {X 0,Y 249.243,Z 756.25,A -85,B 0,C 180,E1 -18883.622,E2 -18883.622} C_VEL
LIN {X 0,Y 249.254,Z 756.22,A -85,B 0,C 180,E1 -18888.617,E2 -18888.617} C_VEL
LIN {X 0,Y 249.471,Z 756.22,A -85,B 0,C 180,E1 -18891.903,E2 -18891.903} C_VEL
LIN {X 0,Y 249.436,Z 756.193,A -85,B 0,C 180,E1 -18896.77,E2 -18896.77} C_VEL
LIN {X 0,Y 249.73,Z 756.175,A -85,B 0,C 180,E1 -18900,E2 -18900} C_VEL
LIN {X 0,Y 249.443,Z 756.223,A -85,B 0,C 180,E1 -18903.23,E2 -18903.23} C_VEL
LIN {X 0,Y 249.483,Z 756.185,A -85,B 0,C 180,E1 -18908.097,E2 -18908.097} C_VEL
LIN {X 0,Y 249.253,Z 756.248,A -85,B 0,C 180,E1 -18911.384,E2 -18911.384} C_VEL
LIN {X 0,Y 249.197,Z 756.229,A -85,B 0,C 180,E1 -18916.381,E2 -18916.381} C_VEL
LIN {X 0,Y 249.082,Z 756.27,A -85,B 0,C 180,E1 -18921.519,E2 -18921.519} C_VEL
LIN {X 0,Y 249.118,Z 756.24,A -85,B 0,C 180,E1 -18925.475,E2 -18925.475} C_VEL
LIN {X 0,Y 249.074,Z 756.269,A -85,B 0,C 180,E1 -18928.989,E2 -18928.989} C_VEL
LIN {X 0,Y 249.032,Z 756.262,A -85,B 0,C 180,E1 -18932.426,E2 -18932.426} C_VEL
LIN {X 0,Y 249.055,Z 756.273,A -85,B 0,C 180,E1 -18936.341,E2 -18936.341} C_VEL
LIN {X 0,Y 248.993,Z 756.238,A -85,B 0,C 180,E1 -18940.481,E2 -18940.481} C_VEL
LIN {X 0,Y 249.002,Z 756.218,A -85,B 0,C 180,E1 -18942.79,E2 -18942.79} C_VEL
LIN {X 0,Y 249.017,Z 756.28,A -85,B 0,C 180,E1 -18947.363,E2 -18947.363} C_VEL
LIN {X 0,Y 249.044,Z 756.242,A -85,B 0,C 180,E1 -18952.2,E2 -18952.2} C_VEL
LIN {X 0,Y 249.045,Z 756.279,A -85,B 0,C 180,E1 -18955.64,E2 -18955.64} C_VEL
LIN {X 0,Y 249.003,Z 756.265,A -85,B 0,C 180,E1 -18959.466,E2 -18959.466} C_VEL
LIN {X 0,Y 249.103,Z 756.42,A -85,B 0,C 180,E1 -18962.939,E2 -18962.939} C_VEL
LIN {X 0,Y 249.732,Z 759.345,A -85,B 0,C 180,E1 -18964.35,E2 -18964.35} C_VEL
LIN {X 0,Y 251.243,Z 763.152,A -85,B 0,C 180,E1 -18964.724,E2 -18964.724} C_VEL
LIN {X 0,Y 257.744,Z 780.085,A -85,B 0,C 180,E1 -18965.92,E2 -18965.92} C_VEL
LIN {X 0,Y 259.858,Z 791.201,A -85,B 0,C 180,E1 -18966.46,E2 -18966.46} C_VEL
LIN {X 0,Y 258.682,Z 834.855,A -85,B 0,C 180,E1 -18967.683,E2 -18967.683} C_VEL
LIN {X 0,Y 258.287,Z 844.074,A -85,B 0,C 180,E1 -18968.134,E2 -18968.134} C_VEL
LIN {X 0,Y 257.462,Z 853.563,A -85,B 0,C 180,E1 -18968.796,E2 -18968.796} C_VEL
LIN {X 0,Y 256.519,Z 861.672,A -85,B 0,C 180,E1 -18969.554,E2 -18969.554} C_VEL
LIN {X 0,Y 255.416,Z 871.222,A -85,B 0,C 180,E1 -18970.72,E2 -18970.72} C_VEL
LIN {X 0,Y 253.79,Z 880.979,A -85,B 0,C 180,E1 -18972.265,E2 -18972.265} C_VEL
LIN {X 0,Y 252.517,Z 888.689,A -85,B 0,C 180,E1 -18973.84,E2 -18973.84} C_VEL
LIN {X 0,Y 251.244,Z 895.03,A -85,B 0,C 180,E1 -18975.419,E2 -18975.419} C_VEL
LIN {X 0,Y 250.22,Z 900.297,A -85,B 0,C 180,E1 -18977.015,E2 -18977.015} C_VEL
LIN {X 0,Y 249.321,Z 904.693,A -85,B 0,C 180,E1 -18978.62,E2 -18978.62} C_VEL
LIN {X 0,Y 248.365,Z 909.859,A -85,B 0,C 180,E1 -18981.046,E2 -18981.046} C_VEL
LIN {X 0,Y 247.673,Z 913.397,A -85,B 0,C 180,E1 -18983.299,E2 -18983.299} C_VEL
LIN {X 0,Y 247.355,Z 915.409,A -85,B 0,C 180,E1 -18985.11,E2 -18985.11} C_VEL
LIN {X 0,Y 247.146,Z 916.674,A -85,B 0,C 180,E1 -18986.74,E2 -18986.74} C_VEL
LIN {X 0,Y 247.035,Z 917.47,A -85,B 0,C 180,E1 -18988.37,E2 -18988.37} C_VEL
LIN {X 0,Y 246.993,Z 917.774,A -85,B 0,C 180,E1 -18990,E2 -18990} C_VEL
LIN {X 0,Y 247.032,Z 917.494,A -85,B 0,C 180,E1 -18991.63,E2 -18991.63} C_VEL
LIN {X 0,Y 247.14,Z 916.746,A -85,B 0,C 180,E1 -18993.26,E2 -18993.26} C_VEL
LIN {X 0,Y 247.35,Z 915.531,A -85,B 0,C 180,E1 -18994.89,E2 -18994.89} C_VEL
LIN {X 0,Y 247.849,Z 912.682,A -85,B 0,C 180,E1 -18997.33,E2 -18997.33} C_VEL
LIN {X 0,Y 248.288,Z 910.087,A -85,B 0,C 180,E1 -18998.956,E2 -18998.956} C_VEL
LIN {X 0,Y 249.257,Z 904.981,A -85,B 0,C 180,E1 -19001.383,E2 -19001.383} C_VEL
LIN {X 0,Y 250.402,Z 899.483,A -85,B 0,C 180,E1 -19003.388,E2 -19003.388} C_VEL
LIN {X 0,Y 251.825,Z 892.569,A -85,B 0,C 180,E1 -19005.375,E2 -19005.375} C_VEL
LIN {X 0,Y 253.172,Z 884.632,A -85,B 0,C 180,E1 -19007.154,E2 -19007.154} C_VEL
LIN {X 0,Y 254.449,Z 877.06,A -85,B 0,C 180,E1 -19008.52,E2 -19008.52} C_VEL
LIN {X 0,Y 255.717,Z 869.115,A -85,B 0,C 180,E1 -19009.674,E2 -19009.674} C_VEL
LIN {X 0,Y 256.768,Z 860.905,A -85,B 0,C 180,E1 -19010.634,E2 -19010.634} C_VEL
LIN {X 0,Y 257.681,Z 852.763,A -85,B 0,C 180,E1 -19011.378,E2 -19011.378} C_VEL
LIN {X 0,Y 258.289,Z 844.097,A -85,B 0,C 180,E1 -19011.989,E2 -19011.989} C_VEL
LIN {X 0,Y 258.754,Z 834.881,A -85,B 0,C 180,E1 -19012.434,E2 -19012.434} C_VEL
LIN {X 0,Y 259.874,Z 790.675,A -85,B 0,C 180,E1 -19013.679,E2 -19013.679} C_VEL
LIN {X 0,Y 257.646,Z 779.695,A -85,B 0,C 180,E1 -19014.227,E2 -19014.227} C_VEL
LIN {X 0,Y 251.935,Z 764.823,A -85,B 0,C 180,E1 -19015.277,E2 -19015.277} C_VEL
LIN {X 0,Y 249.823,Z 759.588,A -85,B 0,C 180,E1 -19015.726,E2 -19015.726} C_VEL
LIN {X 0,Y 249.483,Z 758.247,A -85,B 0,C 180,E1 -19016.222,E2 -19016.222} C_VEL
LIN {X 0,Y 249.107,Z 756.355,A -85,B 0,C 180,E1 -19017.288,E2 -19017.288} C_VEL
LIN {X 0,Y 249.028,Z 756.257,A -85,B 0,C 180,E1 -19022.426,E2 -19022.426} C_VEL
LIN {X 0,Y 249.049,Z 756.263,A -85,B 0,C 180,E1 -19026.342,E2 -19026.342} C_VEL
LIN {X 0,Y 249.007,Z 756.263,A -85,B 0,C 180,E1 -19030.478,E2 -19030.478} C_VEL
LIN {X 0,Y 249.011,Z 756.281,A -85,B 0,C 180,E1 -19032.792,E2 -19032.792} C_VEL
LIN {X 0,Y 249.01,Z 756.217,A -85,B 0,C 180,E1 -19037.361,E2 -19037.361} C_VEL
LIN {X 0,Y 249.049,Z 756.271,A -85,B 0,C 180,E1 -19042.199,E2 -19042.199} C_VEL
LIN {X 0,Y 249.046,Z 756.261,A -85,B 0,C 180,E1 -19045.64,E2 -19045.64} C_VEL
LIN {X 0,Y 249.049,Z 756.275,A -85,B 0,C 180,E1 -19049.473,E2 -19049.473} C_VEL
LIN {X 0,Y 249.069,Z 756.251,A -85,B 0,C 180,E1 -19053.162,E2 -19053.162} C_VEL
LIN {X 0,Y 249.063,Z 756.265,A -85,B 0,C 180,E1 -19056.731,E2 -19056.731} C_VEL
LIN {X 0,Y 249.105,Z 756.262,A -85,B 0,C 180,E1 -19060.211,E2 -19060.211} C_VEL
LIN {X 0,Y 249.197,Z 756.229,A -85,B 0,C 180,E1 -19063.619,E2 -19063.619} C_VEL
LIN {X 0,Y 249.253,Z 756.248,A -85,B 0,C 180,E1 -19068.616,E2 -19068.616} C_VEL
LIN {X 0,Y 249.486,Z 756.185,A -85,B 0,C 180,E1 -19071.903,E2 -19071.903} C_VEL
LIN {X 0,Y 249.443,Z 756.223,A -85,B 0,C 180,E1 -19076.77,E2 -19076.77} C_VEL
LIN {X 0,Y 249.73,Z 756.175,A -85,B 0,C 180,E1 -19080,E2 -19080} C_VEL
LIN {X 0,Y 249.436,Z 756.193,A -85,B 0,C 180,E1 -19083.23,E2 -19083.23} C_VEL
LIN {X 0,Y 249.471,Z 756.22,A -85,B 0,C 180,E1 -19088.097,E2 -19088.097} C_VEL
LIN {X 0,Y 249.254,Z 756.22,A -85,B 0,C 180,E1 -19091.383,E2 -19091.383} C_VEL
LIN {X 0,Y 249.243,Z 756.25,A -85,B 0,C 180,E1 -19096.378,E2 -19096.378} C_VEL
LIN {X 0,Y 249.208,Z 756.253,A -85,B 0,C 180,E1 -19096.604,E2 -19096.604} C_VEL
LIN {X 0,Y 248.43,Z 756.35,A -85,B 0,C 180,E1 -19097.952,E2 -19097.952} C_VEL
LIN {X 0,Y 245.474,Z 756.697,A -85,B 0,C 180,E1 -19100.148,E2 -19100.148} C_VEL
LIN {X 0,Y 243.062,Z 756.994,A -85,B 0,C 180,E1 -19101.937,E2 -19101.937} C_VEL
LIN {X 0,Y 242.091,Z 757.13,A -85,B 0,C 180,E1 -19103.326,E2 -19103.326} C_VEL
LIN {X 0,Y 242.043,Z 757.137,A -85,B 0,C 180,E1 -19103.797,E2 -19103.797} C_VEL
LIN {X 0,Y 242.003,Z 757.14,A -85,B 0,C 180,E1 -19107.688,E2 -19107.688} C_VEL
LIN {X 0,Y 241.975,Z 757.149,A -85,B 0,C 180,E1 -19111.52,E2 -19111.52} C_VEL
LIN {X 0,Y 242.029,Z 757.129,A -85,B 0,C 180,E1 -19115.604,E2 -19115.604} C_VEL
LIN {X 0,Y 241.981,Z 757.084,A -85,B 0,C 180,E1 -19119.714,E2 -19119.714} C_VEL
LIN {X 0,Y 241.936,Z 757.159,A -85,B 0,C 180,E1 -19124.201,E2 -19124.201} C_VEL
LIN {X 0,Y 241.943,Z 757.131,A -85,B 0,C 180,E1 -19128.079,E2 -19128.079} C_VEL
LIN {X 0,Y 242.002,Z 757.149,A -85,B 0,C 180,E1 -19132.42,E2 -19132.42} C_VEL
LIN {X 0,Y 242.051,Z 757.247,A -85,B 0,C 180,E1 -19136.826,E2 -19136.826} C_VEL
LIN {X 0,Y 243.882,Z 766.107,A -85,B 0,C 180,E1 -19141.139,E2 -19141.139} C_VEL
LIN {X 0,Y 245.008,Z 772.002,A -85,B 0,C 180,E1 -19143.741,E2 -19143.741} C_VEL
LIN {X 0,Y 247.303,Z 778.677,A -85,B 0,C 180,E1 -19144.28,E2 -19144.28} C_VEL
LIN {X 0,Y 250.892,Z 799.965,A -85,B 0,C 180,E1 -19145.328,E2 -19145.328} C_VEL
LIN {X 0,Y 252.845,Z 815.419,A -85,B 0,C 180,E1 -19146,E2 -19146} C_VEL
LIN {X 0,Y 251.818,Z 849.723,A -85,B 0,C 180,E1 -19147,E2 -19147} C_VEL
LIN {X 0,Y 250.986,Z 861.142,A -85,B 0,C 180,E1 -19147.591,E2 -19147.591} C_VEL
LIN {X 0,Y 249.748,Z 872.545,A -85,B 0,C 180,E1 -19148.542,E2 -19148.542} C_VEL
LIN {X 0,Y 248.575,Z 881.233,A -85,B 0,C 180,E1 -19149.52,E2 -19149.52} C_VEL
LIN {X 0,Y 247.291,Z 889.536,A -85,B 0,C 180,E1 -19150.708,E2 -19150.708} C_VEL
LIN {X 0,Y 245.871,Z 897.397,A -85,B 0,C 180,E1 -19152.105,E2 -19152.105} C_VEL
LIN {X 0,Y 244.43,Z 904.749,A -85,B 0,C 180,E1 -19153.72,E2 -19153.72} C_VEL
LIN {X 0,Y 242.955,Z 912.212,A -85,B 0,C 180,E1 -19155.766,E2 -19155.766} C_VEL
LIN {X 0,Y 241.588,Z 919.028,A -85,B 0,C 180,E1 -19158.25,E2 -19158.25} C_VEL
LIN {X 0,Y 240.666,Z 924.211,A -85,B 0,C 180,E1 -19160.758,E2 -19160.758} C_VEL
LIN {X 0,Y 240.098,Z 928.018,A -85,B 0,C 180,E1 -19163.276,E2 -19163.276} C_VEL
LIN {X 0,Y 239.88,Z 929.769,A -85,B 0,C 180,E1 -19164.958,E2 -19164.958} C_VEL
LIN {X 0,Y 239.813,Z 931.024,A -85,B 0,C 180,E1 -19166.64,E2 -19166.64} C_VEL
LIN {X 0,Y 239.844,Z 931.805,A -85,B 0,C 180,E1 -19168.321,E2 -19168.321} C_VEL
LIN {X 0,Y 239.892,Z 932.101,A -85,B 0,C 180,E1 -19170,E2 -19170} C_VEL
LIN {X 0,Y 239.844,Z 931.798,A -85,B 0,C 180,E1 -19171.679,E2 -19171.679} C_VEL
LIN {X 0,Y 239.813,Z 931.004,A -85,B 0,C 180,E1 -19173.36,E2 -19173.36} C_VEL
LIN {X 0,Y 239.88,Z 929.735,A -85,B 0,C 180,E1 -19175.042,E2 -19175.042} C_VEL
LIN {X 0,Y 240.234,Z 926.811,A -85,B 0,C 180,E1 -19177.565,E2 -19177.565} C_VEL
LIN {X 0,Y 240.666,Z 924.149,A -85,B 0,C 180,E1 -19179.242,E2 -19179.242} C_VEL
LIN {X 0,Y 241.582,Z 918.947,A -85,B 0,C 180,E1 -19181.75,E2 -19181.75} C_VEL
LIN {X 0,Y 242.955,Z 912.095,A -85,B 0,C 180,E1 -19184.234,E2 -19184.234} C_VEL
LIN {X 0,Y 244.423,Z 904.611,A -85,B 0,C 180,E1 -19186.281,E2 -19186.281} C_VEL
LIN {X 0,Y 245.857,Z 897.234,A -85,B 0,C 180,E1 -19187.896,E2 -19187.896} C_VEL
LIN {X 0,Y 247.27,Z 889.335,A -85,B 0,C 180,E1 -19189.294,E2 -19189.294} C_VEL
LIN {X 0,Y 248.612,Z 880.986,A -85,B 0,C 180,E1 -19190.477,E2 -19190.477} C_VEL
LIN {X 0,Y 249.929,Z 870.55,A -85,B 0,C 180,E1 -19191.633,E2 -19191.633} C_VEL
LIN {X 0,Y 251.082,Z 859.106,A -85,B 0,C 180,E1 -19192.498,E2 -19192.498} C_VEL
LIN {X 0,Y 251.765,Z 849.795,A -85,B 0,C 180,E1 -19192.966,E2 -19192.966} C_VEL
LIN {X 0,Y 252.697,Z 814.266,A -85,B 0,C 180,E1 -19194.013,E2 -19194.013} C_VEL
LIN {X 0,Y 248.996,Z 788.011,A -85,B 0,C 180,E1 -19195.204,E2 -19195.204} C_VEL
LIN {X 0,Y 246.762,Z 776.91,A -85,B 0,C 180,E1 -19195.797,E2 -19195.797} C_VEL
LIN {X 0,Y 245.012,Z 771.919,A -85,B 0,C 180,E1 -19196.236,E2 -19196.236} C_VEL
LIN {X 0,Y 243.67,Z 764.956,A -85,B 0,C 180,E1 -19199.362,E2 -19199.362} C_VEL
LIN {X 0,Y 242.029,Z 757.182,A -85,B 0,C 180,E1 -19203.239,E2 -19203.239} C_VEL
LIN {X 0,Y 242.002,Z 757.15,A -85,B 0,C 180,E1 -19207.58,E2 -19207.58} C_VEL
LIN {X 0,Y 241.943,Z 757.132,A -85,B 0,C 180,E1 -19211.921,E2 -19211.921} C_VEL
LIN {X 0,Y 241.942,Z 757.15,A -85,B 0,C 180,E1 -19216.569,E2 -19216.569} C_VEL
LIN {X 0,Y 241.981,Z 757.083,A -85,B 0,C 180,E1 -19220.286,E2 -19220.286} C_VEL
LIN {X 0,Y 242.037,Z 757.132,A -85,B 0,C 180,E1 -19224.498,E2 -19224.498} C_VEL
LIN {X 0,Y 241.975,Z 757.148,A -85,B 0,C 180,E1 -19228.48,E2 -19228.48} C_VEL
LIN {X 0,Y 242.003,Z 757.141,A -85,B 0,C 180,E1 -19232.312,E2 -19232.312} C_VEL
LIN {X 0,Y 242.059,Z 757.137,A -85,B 0,C 180,E1 -19236.016,E2 -19236.016} C_VEL
LIN {X 0,Y 242.039,Z 757.123,A -85,B 0,C 180,E1 -19239.608,E2 -19239.608} C_VEL
LIN {X 0,Y 242.164,Z 757.131,A -85,B 0,C 180,E1 -19243.278,E2 -19243.278} C_VEL
LIN {X 0,Y 242.188,Z 757.097,A -85,B 0,C 180,E1 -19248.28,E2 -19248.28} C_VEL
LIN {X 0,Y 242.419,Z 757.098,A -85,B 0,C 180,E1 -19251.665,E2 -19251.665} C_VEL
LIN {X 0,Y 242.26,Z 757.108,A -85,B 0,C 180,E1 -19255.007,E2 -19255.007} C_VEL
LIN {X 0,Y 242.638,Z 757.038,A -85,B 0,C 180,E1 -19258.34,E2 -19258.34} C_VEL
LIN {X 0,Y 242.641,Z 757.069,A -85,B 0,C 180,E1 -19261.66,E2 -19261.66} C_VEL
LIN {X 0,Y 242.432,Z 757.065,A -85,B 0,C 180,E1 -19266.706,E2 -19266.706} C_VEL
LIN {X 0,Y 242.316,Z 757.101,A -85,B 0,C 180,E1 -19270.022,E2 -19270.022} C_VEL
LIN {X 0,Y 242.138,Z 757.12,A -85,B 0,C 180,E1 -19275.143,E2 -19275.143} C_VEL
LIN {X 0,Y 242.055,Z 757.124,A -85,B 0,C 180,E1 -19278.626,E2 -19278.626} C_VEL
LIN {X 0,Y 242.006,Z 757.151,A -85,B 0,C 180,E1 -19282.181,E2 -19282.181} C_VEL
LIN {X 0,Y 242.068,Z 757.117,A -85,B 0,C 180,E1 -19285.838,E2 -19285.838} C_VEL
LIN {X 0,Y 242.009,Z 757.152,A -85,B 0,C 180,E1 -19289.583,E2 -19289.583} C_VEL
LIN {X 0,Y 241.983,Z 757.135,A -85,B 0,C 180,E1 -19293.493,E2 -19293.493} C_VEL
LIN {X 0,Y 241.995,Z 757.152,A -85,B 0,C 180,E1 -19297.581,E2 -19297.581} C_VEL
LIN {X 0,Y 241.931,Z 757.099,A -85,B 0,C 180,E1 -19301.924,E2 -19301.924} C_VEL
LIN {X 0,Y 241.934,Z 757.157,A -85,B 0,C 180,E1 -19306.572,E2 -19306.572} C_VEL
LIN {X 0,Y 241.957,Z 757.131,A -85,B 0,C 180,E1 -19310.281,E2 -19310.281} C_VEL
LIN {X 0,Y 241.989,Z 757.153,A -85,B 0,C 180,E1 -19314.489,E2 -19314.489} C_VEL
LIN {X 0,Y 241.953,Z 757.136,A -85,B 0,C 180,E1 -19318.477,E2 -19318.477} C_VEL
LIN {X 0,Y 242.05,Z 757.312,A -85,B 0,C 180,E1 -19322.428,E2 -19322.428} C_VEL
LIN {X 0,Y 242.546,Z 759.599,A -85,B 0,C 180,E1 -19323.535,E2 -19323.535} C_VEL
LIN {X 0,Y 244.346,Z 764.032,A -85,B 0,C 180,E1 -19323.979,E2 -19323.979} C_VEL
LIN {X 0,Y 251.011,Z 780.797,A -85,B 0,C 180,E1 -19325.246,E2 -19325.246} C_VEL
LIN {X 0,Y 252.427,Z 786.638,A -85,B 0,C 180,E1 -19325.575,E2 -19325.575} C_VEL
LIN {X 0,Y 253.344,Z 793.158,A -85,B 0,C 180,E1 -19325.869,E2 -19325.869} C_VEL
LIN {X 0,Y 252.147,Z 835.118,A -85,B 0,C 180,E1 -19327.074,E2 -19327.074} C_VEL
LIN {X 0,Y 251.728,Z 844.345,A -85,B 0,C 180,E1 -19327.537,E2 -19327.537} C_VEL
LIN {X 0,Y 250.852,Z 854.002,A -85,B 0,C 180,E1 -19328.229,E2 -19328.229} C_VEL
LIN {X 0,Y 249.88,Z 861.887,A -85,B 0,C 180,E1 -19328.986,E2 -19328.986} C_VEL
LIN {X 0,Y 248.746,Z 871.435,A -85,B 0,C 180,E1 -19330.181,E2 -19330.181} C_VEL
LIN {X 0,Y 247.045,Z 881.191,A -85,B 0,C 180,E1 -19331.764,E2 -19331.764} C_VEL
LIN {X 0,Y 245.7,Z 888.901,A -85,B 0,C 180,E1 -19333.379,E2 -19333.379} C_VEL
LIN {X 0,Y 244.387,Z 895.241,A -85,B 0,C 180,E1 -19335,E2 -19335} C_VEL
LIN {X 0,Y 243.325,Z 900.507,A -85,B 0,C 180,E1 -19336.64,E2 -19336.64} C_VEL
LIN {X 0,Y 242.376,Z 904.903,A -85,B 0,C 180,E1 -19338.289,E2 -19338.289} C_VEL
LIN {X 0,Y 241.345,Z 910.07,A -85,B 0,C 180,E1 -19340.784,E2 -19340.784} C_VEL
LIN {X 0,Y 240.804,Z 912.719,A -85,B 0,C 180,E1 -19342.453,E2 -19342.453} C_VEL
LIN {X 0,Y 240.281,Z 915.619,A -85,B 0,C 180,E1 -19344.966,E2 -19344.966} C_VEL
LIN {X 0,Y 240.07,Z 916.883,A -85,B 0,C 180,E1 -19346.643,E2 -19346.643} C_VEL
LIN {X 0,Y 239.947,Z 917.679,A -85,B 0,C 180,E1 -19348.322,E2 -19348.322} C_VEL
LIN {X 0,Y 239.924,Z 917.982,A -85,B 0,C 180,E1 -19350,E2 -19350} C_VEL
LIN {X 0,Y 239.945,Z 917.703,A -85,B 0,C 180,E1 -19351.678,E2 -19351.678} C_VEL
LIN {X 0,Y 240.065,Z 916.954,A -85,B 0,C 180,E1 -19353.357,E2 -19353.357} C_VEL
LIN {X 0,Y 240.274,Z 915.739,A -85,B 0,C 180,E1 -19355.034,E2 -19355.034} C_VEL
LIN {X 0,Y 240.802,Z 912.889,A -85,B 0,C 180,E1 -19357.547,E2 -19357.547} C_VEL
LIN {X 0,Y 241.286,Z 910.294,A -85,B 0,C 180,E1 -19359.218,E2 -19359.218} C_VEL
LIN {X 0,Y 242.295,Z 905.189,A -85,B 0,C 180,E1 -19361.715,E2 -19361.715} C_VEL
LIN {X 0,Y 243.493,Z 899.69,A -85,B 0,C 180,E1 -19363.776,E2 -19363.776} C_VEL
LIN {X 0,Y 244.994,Z 892.775,A -85,B 0,C 180,E1 -19365.814,E2 -19365.814} C_VEL
LIN {X 0,Y 246.42,Z 884.837,A -85,B 0,C 180,E1 -19367.64,E2 -19367.64} C_VEL
LIN {X 0,Y 247.749,Z 877.264,A -85,B 0,C 180,E1 -19369.04,E2 -19369.04} C_VEL
LIN {X 0,Y 249.049,Z 869.319,A -85,B 0,C 180,E1 -19370.224,E2 -19370.224} C_VEL
LIN {X 0,Y 250.152,Z 861.107,A -85,B 0,C 180,E1 -19371.206,E2 -19371.206} C_VEL
LIN {X 0,Y 251.152,Z 852.139,A -85,B 0,C 180,E1 -19372.036,E2 -19372.036} C_VEL
LIN {X 0,Y 251.852,Z 842.466,A -85,B 0,C 180,E1 -19372.7,E2 -19372.7} C_VEL
LIN {X 0,Y 252.388,Z 830.861,A -85,B 0,C 180,E1 -19373.206,E2 -19373.206} C_VEL
LIN {X 0,Y 253.312,Z 791.503,A -85,B 0,C 180,E1 -19374.312,E2 -19374.312} C_VEL
LIN {X 0,Y 251.538,Z 782.36,A -85,B 0,C 180,E1 -19374.778,E2 -19374.778} C_VEL
LIN {X 0,Y 245.944,Z 767.719,A -85,B 0,C 180,E1 -19375.851,E2 -19375.851} C_VEL
LIN {X 0,Y 242.62,Z 759.789,A -85,B 0,C 180,E1 -19376.554,E2 -19376.554} C_VEL
LIN {X 0,Y 242.399,Z 758.886,A -85,B 0,C 180,E1 -19376.857,E2 -19376.857} C_VEL
LIN {X 0,Y 242.038,Z 757.241,A -85,B 0,C 180,E1 -19377.801,E2 -19377.801} C_VEL
LIN {X 0,Y 241.989,Z 757.135,A -85,B 0,C 180,E1 -19382.623,E2 -19382.623} C_VEL
LIN {X 0,Y 242.007,Z 757.152,A -85,B 0,C 180,E1 -19385.596,E2 -19385.596} C_VEL
LIN {X 0,Y 241.957,Z 757.129,A -85,B 0,C 180,E1 -19389.719,E2 -19389.719} C_VEL
LIN {X 0,Y 241.927,Z 757.148,A -85,B 0,C 180,E1 -19394.203,E2 -19394.203} C_VEL
LIN {X 0,Y 241.931,Z 757.099,A -85,B 0,C 180,E1 -19398.076,E2 -19398.076} C_VEL
LIN {X 0,Y 241.995,Z 757.151,A -85,B 0,C 180,E1 -19402.419,E2 -19402.419} C_VEL
LIN {X 0,Y 241.983,Z 757.135,A -85,B 0,C 180,E1 -19406.507,E2 -19406.507} C_VEL
LIN {X 0,Y 242.015,Z 757.152,A -85,B 0,C 180,E1 -19410.597,E2 -19410.597} C_VEL
LIN {X 0,Y 242.069,Z 757.117,A -85,B 0,C 180,E1 -19414.183,E2 -19414.183} C_VEL
LIN {X 0,Y 242.028,Z 757.148,A -85,B 0,C 180,E1 -19418.313,E2 -19418.313} C_VEL
LIN {X 0,Y 242.117,Z 757.108,A -85,B 0,C 180,E1 -19423.316,E2 -19423.316} C_VEL
LIN {X 0,Y 242.186,Z 757.128,A -85,B 0,C 180,E1 -19428.28,E2 -19428.28} C_VEL
LIN {X 0,Y 242.437,Z 757.064,A -85,B 0,C 180,E1 -19431.666,E2 -19431.666} C_VEL
LIN {X 0,Y 242.264,Z 757.107,A -85,B 0,C 180,E1 -19435.007,E2 -19435.007} C_VEL
LIN {X 0,Y 242.641,Z 757.069,A -85,B 0,C 180,E1 -19438.34,E2 -19438.34} C_VEL
LIN {X 0,Y 242.637,Z 757.038,A -85,B 0,C 180,E1 -19441.66,E2 -19441.66} C_VEL
LIN {X 0,Y 242.429,Z 757.098,A -85,B 0,C 180,E1 -19446.659,E2 -19446.659} C_VEL
LIN {X 0,Y 242.314,Z 757.098,A -85,B 0,C 180,E1 -19450.022,E2 -19450.022} C_VEL
LIN {X 0,Y 242.168,Z 757.124,A -85,B 0,C 180,E1 -19455.141,E2 -19455.141} C_VEL
LIN {X 0,Y 242.075,Z 757.136,A -85,B 0,C 180,E1 -19458.624,E2 -19458.624} C_VEL
LIN {X 0,Y 242.014,Z 757.125,A -85,B 0,C 180,E1 -19462.18,E2 -19462.18} C_VEL
LIN {X 0,Y 242.043,Z 757.137,A -85,B 0,C 180,E1 -19463.797,E2 -19463.797} C_VEL
LIN {X 0,Y 241.783,Z 757.18,A -85,B 0,C 180,E1 -19464.725,E2 -19464.725} C_VEL
LIN {X 0,Y 240.463,Z 757.348,A -85,B 0,C 180,E1 -19466.097,E2 -19466.097} C_VEL
LIN {X 0,Y 236.069,Z 757.876,A -85,B 0,C 180,E1 -19469.294,E2 -19469.294} C_VEL
LIN {X 0,Y 234.992,Z 758.009,A -85,B 0,C 180,E1 -19470.728,E2 -19470.728} C_VEL
LIN {X 0,Y 234.904,Z 758.021,A -85,B 0,C 180,E1 -19471.215,E2 -19471.215} C_VEL
LIN {X 0,Y 234.961,Z 758.022,A -85,B 0,C 180,E1 -19474.633,E2 -19474.633} C_VEL
LIN {X 0,Y 234.942,Z 757.96,A -85,B 0,C 180,E1 -19478.944,E2 -19478.944} C_VEL
LIN {X 0,Y 234.92,Z 758.026,A -85,B 0,C 180,E1 -19483.478,E2 -19483.478} C_VEL
LIN {X 0,Y 234.888,Z 758.026,A -85,B 0,C 180,E1 -19486.514,E2 -19486.514} C_VEL
LIN {X 0,Y 234.955,Z 758.026,A -85,B 0,C 180,E1 -19491.086,E2 -19491.086} C_VEL
LIN {X 0,Y 234.974,Z 758.019,A -85,B 0,C 180,E1 -19495.369,E2 -19495.369} C_VEL
LIN {X 0,Y 235.013,Z 758.215,A -85,B 0,C 180,E1 -19496.294,E2 -19496.294} C_VEL
LIN {X 0,Y 236.837,Z 766.944,A -85,B 0,C 180,E1 -19500.684,E2 -19500.684} C_VEL
LIN {X 0,Y 237.772,Z 771.802,A -85,B 0,C 180,E1 -19502.882,E2 -19502.882} C_VEL
LIN {X 0,Y 241.103,Z 780.881,A -85,B 0,C 180,E1 -19503.645,E2 -19503.645} C_VEL
LIN {X 0,Y 244.583,Z 801.73,A -85,B 0,C 180,E1 -19504.709,E2 -19504.709} C_VEL
LIN {X 0,Y 246.353,Z 816.072,A -85,B 0,C 180,E1 -19505.353,E2 -19505.353} C_VEL
LIN {X 0,Y 245.307,Z 849.53,A -85,B 0,C 180,E1 -19506.353,E2 -19506.353} C_VEL
LIN {X 0,Y 244.488,Z 860.533,A -85,B 0,C 180,E1 -19506.933,E2 -19506.933} C_VEL
LIN {X 0,Y 243.147,Z 872.341,A -85,B 0,C 180,E1 -19507.929,E2 -19507.929} C_VEL
LIN {X 0,Y 241.937,Z 881.029,A -85,B 0,C 180,E1 -19508.932,E2 -19508.932} C_VEL
LIN {X 0,Y 240.592,Z 889.331,A -85,B 0,C 180,E1 -19510.149,E2 -19510.149} C_VEL
LIN {X 0,Y 239.13,Z 897.191,A -85,B 0,C 180,E1 -19511.582,E2 -19511.582} C_VEL
LIN {X 0,Y 237.625,Z 904.543,A -85,B 0,C 180,E1 -19513.24,E2 -19513.24} C_VEL
LIN {X 0,Y 236.04,Z 912.004,A -85,B 0,C 180,E1 -19515.34,E2 -19515.34} C_VEL
LIN {X 0,Y 234.617,Z 918.819,A -85,B 0,C 180,E1 -19517.896,E2 -19517.896} C_VEL
LIN {X 0,Y 233.647,Z 924.002,A -85,B 0,C 180,E1 -19520.477,E2 -19520.477} C_VEL
LIN {X 0,Y 233.05,Z 927.81,A -85,B 0,C 180,E1 -19523.072,E2 -19523.072} C_VEL
LIN {X 0,Y 232.783,Z 929.815,A -85,B 0,C 180,E1 -19525.075,E2 -19525.075} C_VEL
LIN {X 0,Y 232.757,Z 931.596,A -85,B 0,C 180,E1 -19528.27,E2 -19528.27} C_VEL
LIN {X 0,Y 232.803,Z 931.892,A -85,B 0,C 180,E1 -19530,E2 -19530} C_VEL
LIN {X 0,Y 232.757,Z 931.59,A -85,B 0,C 180,E1 -19531.73,E2 -19531.73} C_VEL
LIN {X 0,Y 232.763,Z 929.835,A -85,B 0,C 180,E1 -19534.867,E2 -19534.867} C_VEL
LIN {X 0,Y 233.052,Z 927.761,A -85,B 0,C 180,E1 -19536.928,E2 -19536.928} C_VEL
LIN {X 0,Y 233.646,Z 923.938,A -85,B 0,C 180,E1 -19539.523,E2 -19539.523} C_VEL
LIN {X 0,Y 234.611,Z 918.736,A -85,B 0,C 180,E1 -19542.104,E2 -19542.104} C_VEL
LIN {X 0,Y 236.039,Z 911.883,A -85,B 0,C 180,E1 -19544.66,E2 -19544.66} C_VEL
LIN {X 0,Y 237.616,Z 904.4,A -85,B 0,C 180,E1 -19546.761,E2 -19546.761} C_VEL
LIN {X 0,Y 239.111,Z 897.022,A -85,B 0,C 180,E1 -19548.419,E2 -19548.419} C_VEL
LIN {X 0,Y 240.565,Z 889.122,A -85,B 0,C 180,E1 -19549.854,E2 -19549.854} C_VEL
LIN {X 0,Y 241.971,Z 880.772,A -85,B 0,C 180,E1 -19551.065,E2 -19551.065} C_VEL
LIN {X 0,Y 243.312,Z 870.579,A -85,B 0,C 180,E1 -19552.225,E2 -19552.225} C_VEL
LIN {X 0,Y 244.561,Z 858.888,A -85,B 0,C 180,E1 -19553.132,E2 -19553.132} C_VEL
LIN {X 0,Y 245.249,Z 849.785,A -85,B 0,C 180,E1 -19553.603,E2 -19553.603} C_VEL
LIN {X 0,Y 246.109,Z 820.483,A -85,B 0,C 180,E1 -19554.495,E2 -19554.495} C_VEL
LIN {X 0,Y 246.103,Z 813.864,A -85,B 0,C 180,E1 -19554.704,E2 -19554.704} C_VEL
LIN {X 0,Y 242.444,Z 788.411,A -85,B 0,C 180,E1 -19555.915,E2 -19555.915} C_VEL
LIN {X 0,Y 240.704,Z 779.652,A -85,B 0,C 180,E1 -19556.399,E2 -19556.399} C_VEL
LIN {X 0,Y 237.788,Z 771.789,A -85,B 0,C 180,E1 -19557.074,E2 -19557.074} C_VEL
LIN {X 0,Y 236.829,Z 766.841,A -85,B 0,C 180,E1 -19559.317,E2 -19559.317} C_VEL
LIN {X 0,Y 234.99,Z 758.179,A -85,B 0,C 180,E1 -19563.707,E2 -19563.707} C_VEL
LIN {X 0,Y 234.941,Z 758.02,A -85,B 0,C 180,E1 -19566.747,E2 -19566.747} C_VEL
LIN {X 0,Y 234.942,Z 758.026,A -85,B 0,C 180,E1 -19568.945,E2 -19568.945} C_VEL
LIN {X 0,Y 234.888,Z 758.028,A -85,B 0,C 180,E1 -19573.486,E2 -19573.486} C_VEL
LIN {X 0,Y 234.92,Z 758.024,A -85,B 0,C 180,E1 -19576.522,E2 -19576.522} C_VEL
LIN {X 0,Y 234.955,Z 757.958,A -85,B 0,C 180,E1 -19581.086,E2 -19581.086} C_VEL
LIN {X 0,Y 234.961,Z 758.023,A -85,B 0,C 180,E1 -19585.367,E2 -19585.367} C_VEL
LIN {X 0,Y 234.924,Z 758.015,A -85,B 0,C 180,E1 -19589.431,E2 -19589.431} C_VEL
LIN {X 0,Y 234.994,Z 758.025,A -85,B 0,C 180,E1 -19593.794,E2 -19593.794} C_VEL
LIN {X 0,Y 235.013,Z 757.994,A -85,B 0,C 180,E1 -19598.97,E2 -19598.97} C_VEL
LIN {X 0,Y 235.098,Z 758.011,A -85,B 0,C 180,E1 -19603.059,E2 -19603.059} C_VEL
LIN {X 0,Y 235.12,Z 757.975,A -85,B 0,C 180,E1 -19607.922,E2 -19607.922} C_VEL
LIN {X 0,Y 235.37,Z 757.975,A -85,B 0,C 180,E1 -19611.414,E2 -19611.414} C_VEL
LIN {X 0,Y 235.4,Z 757.973,A -85,B 0,C 180,E1 -19613.141,E2 -19613.141} C_VEL
LIN {X 0,Y 235.598,Z 757.914,A -85,B 0,C 180,E1 -19618.291,E2 -19618.291} C_VEL
LIN {X 0,Y 235.601,Z 757.946,A -85,B 0,C 180,E1 -19621.71,E2 -19621.71} C_VEL
LIN {X 0,Y 235.406,Z 757.938,A -85,B 0,C 180,E1 -19626.859,E2 -19626.859} C_VEL
LIN {X 0,Y 235.239,Z 757.984,A -85,B 0,C 180,E1 -19630.327,E2 -19630.327} C_VEL
LIN {X 0,Y 235.082,Z 757.994,A -85,B 0,C 180,E1 -19635.609,E2 -19635.609} C_VEL
LIN {X 0,Y 234.995,Z 758.008,A -85,B 0,C 180,E1 -19639.207,E2 -19639.207} C_VEL
LIN {X 0,Y 234.953,Z 758.027,A -85,B 0,C 180,E1 -19642.884,E2 -19642.884} C_VEL
LIN {X 0,Y 234.969,Z 758.003,A -85,B 0,C 180,E1 -19646.658,E2 -19646.658} C_VEL
LIN {X 0,Y 234.924,Z 758.034,A -85,B 0,C 180,E1 -19650.569,E2 -19650.569} C_VEL
LIN {X 0,Y 234.935,Z 758.019,A -85,B 0,C 180,E1 -19654.638,E2 -19654.638} C_VEL
LIN {X 0,Y 234.943,Z 758.016,A -85,B 0,C 180,E1 -19658.944,E2 -19658.944} C_VEL
LIN {X 0,Y 234.888,Z 757.984,A -85,B 0,C 180,E1 -19664.103,E2 -19664.103} C_VEL
LIN {X 0,Y 234.884,Z 758.038,A -85,B 0,C 180,E1 -19668.42,E2 -19668.42} C_VEL
LIN {X 0,Y 234.919,Z 758,A -85,B 0,C 180,E1 -19671.079,E2 -19671.079} C_VEL
LIN {X 0,Y 234.931,Z 758.04,A -85,B 0,C 180,E1 -19675.362,E2 -19675.362} C_VEL
LIN {X 0,Y 234.9,Z 758.02,A -85,B 0,C 180,E1 -19679.428,E2 -19679.428} C_VEL
LIN {X 0,Y 234.985,Z 758.249,A -85,B 0,C 180,E1 -19681.897,E2 -19681.897} C_VEL
LIN {X 0,Y 235.399,Z 760.009,A -85,B 0,C 180,E1 -19682.698,E2 -19682.698} C_VEL
LIN {X 0,Y 240.082,Z 770.936,A -85,B 0,C 180,E1 -19683.702,E2 -19683.702} C_VEL
LIN {X 0,Y 245.504,Z 785.338,A -85,B 0,C 180,E1 -19684.79,E2 -19684.79} C_VEL
LIN {X 0,Y 246.895,Z 794.033,A -85,B 0,C 180,E1 -19685.217,E2 -19685.217} C_VEL
LIN {X 0,Y 245.627,Z 835.783,A -85,B 0,C 180,E1 -19686.448,E2 -19686.448} C_VEL
LIN {X 0,Y 245.1,Z 845.515,A -85,B 0,C 180,E1 -19686.959,E2 -19686.959} C_VEL
LIN {X 0,Y 243.982,Z 856.592,A -85,B 0,C 180,E1 -19687.807,E2 -19687.807} C_VEL
LIN {X 0,Y 242.734,Z 867.157,A -85,B 0,C 180,E1 -19689.004,E2 -19689.004} C_VEL
LIN {X 0,Y 241.354,Z 875.533,A -85,B 0,C 180,E1 -19690.214,E2 -19690.214} C_VEL
LIN {X 0,Y 239.944,Z 883.439,A -85,B 0,C 180,E1 -19691.647,E2 -19691.647} C_VEL
LIN {X 0,Y 238.902,Z 889.113,A -85,B 0,C 180,E1 -19692.892,E2 -19692.892} C_VEL
LIN {X 0,Y 237.549,Z 895.452,A -85,B 0,C 180,E1 -19694.558,E2 -19694.558} C_VEL
LIN {X 0,Y 236.438,Z 900.717,A -85,B 0,C 180,E1 -19696.244,E2 -19696.244} C_VEL
LIN {X 0,Y 235.419,Z 905.114,A -85,B 0,C 180,E1 -19697.938,E2 -19697.938} C_VEL
LIN {X 0,Y 234.35,Z 910.279,A -85,B 0,C 180,E1 -19700.506,E2 -19700.506} C_VEL
LIN {X 0,Y 233.766,Z 912.929,A -85,B 0,C 180,E1 -19702.225,E2 -19702.225} C_VEL
LIN {X 0,Y 233.503,Z 914.394,A -85,B 0,C 180,E1 -19703.335,E2 -19703.335} C_VEL
LIN {X 0,Y 232.997,Z 917.091,A -85,B 0,C 180,E1 -19706.541,E2 -19706.541} C_VEL
LIN {X 0,Y 232.862,Z 917.887,A -85,B 0,C 180,E1 -19708.27,E2 -19708.27} C_VEL
LIN {X 0,Y 232.835,Z 918.19,A -85,B 0,C 180,E1 -19710,E2 -19710} C_VEL
LIN {X 0,Y 232.86,Z 917.911,A -85,B 0,C 180,E1 -19711.73,E2 -19711.73} C_VEL
LIN {X 0,Y 232.993,Z 917.162,A -85,B 0,C 180,E1 -19713.459,E2 -19713.459} C_VEL
LIN {X 0,Y 233.5,Z 914.551,A -85,B 0,C 180,E1 -19716.659,E2 -19716.659} C_VEL
LIN {X 0,Y 234.019,Z 911.946,A -85,B 0,C 180,E1 -19718.636,E2 -19718.636} C_VEL
LIN {X 0,Y 234.952,Z 907.297,A -85,B 0,C 180,E1 -19721.211,E2 -19721.211} C_VEL
LIN {X 0,Y 236.118,Z 902.231,A -85,B 0,C 180,E1 -19723.337,E2 -19723.337} C_VEL
LIN {X 0,Y 237.232,Z 897.279,A -85,B 0,C 180,E1 -19725.024,E2 -19725.024} C_VEL
LIN {X 0,Y 238.522,Z 891.3,A -85,B 0,C 180,E1 -19726.695,E2 -19726.695} C_VEL
LIN {X 0,Y 239.858,Z 884.025,A -85,B 0,C 180,E1 -19728.36,E2 -19728.36} C_VEL
LIN {X 0,Y 241.299,Z 876.241,A -85,B 0,C 180,E1 -19729.791,E2 -19729.791} C_VEL
LIN {X 0,Y 242.642,Z 868.024,A -85,B 0,C 180,E1 -19731.004,E2 -19731.004} C_VEL
LIN {X 0,Y 243.998,Z 857.807,A -85,B 0,C 180,E1 -19732.184,E2 -19732.184} C_VEL
LIN {X 0,Y 245.148,Z 845.653,A -85,B 0,C 180,E1 -19733.156,E2 -19733.156} C_VEL
LIN {X 0,Y 245.637,Z 836.473,A -85,B 0,C 180,E1 -19733.651,E2 -19733.651} C_VEL
LIN {X 0,Y 246.648,Z 802.506,A -85,B 0,C 180,E1 -19734.673,E2 -19734.673} C_VEL
LIN {X 0,Y 246.866,Z 792.474,A -85,B 0,C 180,E1 -19734.965,E2 -19734.965} C_VEL
LIN {X 0,Y 245.253,Z 784.283,A -85,B 0,C 180,E1 -19735.402,E2 -19735.402} C_VEL
LIN {X 0,Y 239.069,Z 768.392,A -85,B 0,C 180,E1 -19736.637,E2 -19736.637} C_VEL
LIN {X 0,Y 235.469,Z 760.192,A -85,B 0,C 180,E1 -19737.4,E2 -19737.4} C_VEL
LIN {X 0,Y 235.268,Z 759.402,A -85,B 0,C 180,E1 -19737.616,E2 -19737.616} C_VEL
LIN {X 0,Y 235.002,Z 758.126,A -85,B 0,C 180,E1 -19738.344,E2 -19738.344} C_VEL
LIN {X 0,Y 234.942,Z 758.016,A -85,B 0,C 180,E1 -19743.114,E2 -19743.114} C_VEL
LIN {X 0,Y 234.928,Z 758.012,A -85,B 0,C 180,E1 -19746.749,E2 -19746.749} C_VEL
LIN {X 0,Y 234.943,Z 757.996,A -85,B 0,C 180,E1 -19748.944,E2 -19748.944} C_VEL
LIN {X 0,Y 234.886,Z 758.036,A -85,B 0,C 180,E1 -19753.486,E2 -19753.486} C_VEL
LIN {X 0,Y 234.881,Z 757.98,A -85,B 0,C 180,E1 -19756.512,E2 -19756.512} C_VEL
LIN {X 0,Y 234.918,Z 758.018,A -85,B 0,C 180,E1 -19761.078,E2 -19761.078} C_VEL
LIN {X 0,Y 234.935,Z 758.02,A -85,B 0,C 180,E1 -19765.362,E2 -19765.362} C_VEL
LIN {X 0,Y 234.924,Z 758.034,A -85,B 0,C 180,E1 -19769.431,E2 -19769.431} C_VEL
LIN {X 0,Y 234.995,Z 757.998,A -85,B 0,C 180,E1 -19773.794,E2 -19773.794} C_VEL
LIN {X 0,Y 234.998,Z 758.025,A -85,B 0,C 180,E1 -19778.968,E2 -19778.968} C_VEL
LIN {X 0,Y 235.058,Z 757.986,A -85,B 0,C 180,E1 -19783.092,E2 -19783.092} C_VEL
LIN {X 0,Y 235.116,Z 758.009,A -85,B 0,C 180,E1 -19787.922,E2 -19787.922} C_VEL
LIN {X 0,Y 235.392,Z 757.943,A -85,B 0,C 180,E1 -19791.414,E2 -19791.414} C_VEL
LIN {X 0,Y 235.408,Z 757.938,A -85,B 0,C 180,E1 -19793.141,E2 -19793.141} C_VEL
LIN {X 0,Y 235.601,Z 757.946,A -85,B 0,C 180,E1 -19798.29,E2 -19798.29} C_VEL
LIN {X 0,Y 235.597,Z 757.914,A -85,B 0,C 180,E1 -19801.709,E2 -19801.709} C_VEL
LIN {X 0,Y 235.4,Z 757.973,A -85,B 0,C 180,E1 -19806.859,E2 -19806.859} C_VEL
LIN {X 0,Y 235.239,Z 757.977,A -85,B 0,C 180,E1 -19810.326,E2 -19810.326} C_VEL
LIN {X 0,Y 235.115,Z 758.005,A -85,B 0,C 180,E1 -19815.606,E2 -19815.606} C_VEL
LIN {X 0,Y 235.011,Z 758.01,A -85,B 0,C 180,E1 -19819.205,E2 -19819.205} C_VEL
LIN {X 0,Y 234.962,Z 758.01,A -85,B 0,C 180,E1 -19822.882,E2 -19822.882} C_VEL
LIN {X 0,Y 234.969,Z 758.025,A -85,B 0,C 180,E1 -19826.657,E2 -19826.657} C_VEL
LIN {X 0,Y 234.904,Z 758.021,A -85,B 0,C 180,E1 -19831.215,E2 -19831.215} C_VEL
LIN {X 0,Y 234.237,Z 758.121,A -85,B 0,C 180,E1 -19832.647,E2 -19832.647} C_VEL
LIN {X 0,Y 231.387,Z 758.464,A -85,B 0,C 180,E1 -19834.984,E2 -19834.984} C_VEL
LIN {X 0,Y 228.966,Z 758.731,A -85,B 0,C 180,E1 -19836.89,E2 -19836.89} C_VEL
LIN {X 0,Y 227.929,Z 758.836,A -85,B 0,C 180,E1 -19838.368,E2 -19838.368} C_VEL
LIN {X 0,Y 227.845,Z 758.843,A -85,B 0,C 180,E1 -19838.87,E2 -19838.87} C_VEL
LIN {X 0,Y 227.838,Z 758.894,A -85,B 0,C 180,E1 -19842.736,E2 -19842.736} C_VEL
LIN {X 0,Y 227.814,Z 758.896,A -85,B 0,C 180,E1 -19847.258,E2 -19847.258} C_VEL
LIN {X 0,Y 227.87,Z 758.915,A -85,B 0,C 180,E1 -19851.914,E2 -19851.914} C_VEL
LIN {X 0,Y 227.952,Z 759.045,A -85,B 0,C 180,E1 -19855.627,E2 -19855.627} C_VEL
LIN {X 0,Y 229.667,Z 767.225,A -85,B 0,C 180,E1 -19859.922,E2 -19859.922} C_VEL
LIN {X 0,Y 230.514,Z 771.436,A -85,B 0,C 180,E1 -19861.928,E2 -19861.928} C_VEL
LIN {X 0,Y 232.433,Z 776.619,A -85,B 0,C 180,E1 -19862.445,E2 -19862.445} C_VEL
LIN {X 0,Y 235.093,Z 783.823,A -85,B 0,C 180,E1 -19863.022,E2 -19863.022} C_VEL
LIN {X 0,Y 238.408,Z 804.495,A -85,B 0,C 180,E1 -19864.103,E2 -19864.103} C_VEL
LIN {X 0,Y 239.878,Z 817.115,A -85,B 0,C 180,E1 -19864.681,E2 -19864.681} C_VEL
LIN {X 0,Y 238.833,Z 849.337,A -85,B 0,C 180,E1 -19865.671,E2 -19865.671} C_VEL
LIN {X 0,Y 237.92,Z 861.01,A -85,B 0,C 180,E1 -19866.308,E2 -19866.308} C_VEL
LIN {X 0,Y 236.586,Z 872.138,A -85,B 0,C 180,E1 -19867.283,E2 -19867.283} C_VEL
LIN {X 0,Y 235.335,Z 880.824,A -85,B 0,C 180,E1 -19868.311,E2 -19868.311} C_VEL
LIN {X 0,Y 233.91,Z 889.125,A -85,B 0,C 180,E1 -19869.557,E2 -19869.557} C_VEL
LIN {X 0,Y 232.411,Z 896.985,A -85,B 0,C 180,E1 -19871.03,E2 -19871.03} C_VEL
LIN {X 0,Y 230.836,Z 904.337,A -85,B 0,C 180,E1 -19872.732,E2 -19872.732} C_VEL
LIN {X 0,Y 229.156,Z 911.797,A -85,B 0,C 180,E1 -19874.889,E2 -19874.889} C_VEL
LIN {X 0,Y 227.656,Z 918.611,A -85,B 0,C 180,E1 -19877.52,E2 -19877.52} C_VEL
LIN {X 0,Y 226.617,Z 923.794,A -85,B 0,C 180,E1 -19880.179,E2 -19880.179} C_VEL
LIN {X 0,Y 226,Z 927.602,A -85,B 0,C 180,E1 -19882.854,E2 -19882.854} C_VEL
LIN {X 0,Y 225.695,Z 929.84,A -85,B 0,C 180,E1 -19885.176,E2 -19885.176} C_VEL
LIN {X 0,Y 225.672,Z 931.388,A -85,B 0,C 180,E1 -19888.215,E2 -19888.215} C_VEL
LIN {X 0,Y 225.716,Z 931.683,A -85,B 0,C 180,E1 -19890,E2 -19890} C_VEL
LIN {X 0,Y 225.672,Z 931.381,A -85,B 0,C 180,E1 -19891.785,E2 -19891.785} C_VEL
LIN {X 0,Y 225.673,Z 929.861,A -85,B 0,C 180,E1 -19894.76,E2 -19894.76} C_VEL
LIN {X 0,Y 226.001,Z 927.551,A -85,B 0,C 180,E1 -19897.145,E2 -19897.145} C_VEL
LIN {X 0,Y 226.616,Z 923.727,A -85,B 0,C 180,E1 -19899.821,E2 -19899.821} C_VEL
LIN {X 0,Y 227.651,Z 918.525,A -85,B 0,C 180,E1 -19902.48,E2 -19902.48} C_VEL
LIN {X 0,Y 229.156,Z 911.671,A -85,B 0,C 180,E1 -19905.111,E2 -19905.111} C_VEL
LIN {X 0,Y 230.827,Z 904.188,A -85,B 0,C 180,E1 -19907.269,E2 -19907.269} C_VEL
LIN {X 0,Y 232.38,Z 896.81,A -85,B 0,C 180,E1 -19908.973,E2 -19908.973} C_VEL
LIN {X 0,Y 233.682,Z 890.142,A -85,B 0,C 180,E1 -19910.235,E2 -19910.235} C_VEL
LIN {X 0,Y 235.113,Z 882.062,A -85,B 0,C 180,E1 -19911.48,E2 -19911.48} C_VEL
LIN {X 0,Y 236.325,Z 873.681,A -85,B 0,C 180,E1 -19912.513,E2 -19912.513} C_VEL
LIN {X 0,Y 237.472,Z 864.065,A -85,B 0,C 180,E1 -19913.418,E2 -19913.418} C_VEL
LIN {X 0,Y 238.591,Z 852.894,A -85,B 0,C 180,E1 -19914.143,E2 -19914.143} C_VEL
LIN {X 0,Y 239.195,Z 836.785,A -85,B 0,C 180,E1 -19914.716,E2 -19914.716} C_VEL
LIN {X 0,Y 239.675,Z 814.808,A -85,B 0,C 180,E1 -19915.375,E2 -19915.375} C_VEL
LIN {X 0,Y 236.016,Z 789.242,A -85,B 0,C 180,E1 -19916.64,E2 -19916.64} C_VEL
LIN {X 0,Y 234.469,Z 781.628,A -85,B 0,C 180,E1 -19917.084,E2 -19917.084} C_VEL
LIN {X 0,Y 230.59,Z 771.706,A -85,B 0,C 180,E1 -19917.966,E2 -19917.966} C_VEL
LIN {X 0,Y 229.983,Z 768.727,A -85,B 0,C 180,E1 -19919.271,E2 -19919.271} C_VEL
LIN {X 0,Y 228.161,Z 760.119,A -85,B 0,C 180,E1 -19923.729,E2 -19923.729} C_VEL
LIN {X 0,Y 227.935,Z 758.927,A -85,B 0,C 180,E1 -19924.51,E2 -19924.51} C_VEL
LIN {X 0,Y 227.87,Z 758.915,A -85,B 0,C 180,E1 -19928.086,E2 -19928.086} C_VEL
LIN {X 0,Y 227.814,Z 758.897,A -85,B 0,C 180,E1 -19932.742,E2 -19932.742} C_VEL
LIN {X 0,Y 227.838,Z 758.891,A -85,B 0,C 180,E1 -19937.264,E2 -19937.264} C_VEL
LIN {X 0,Y 227.872,Z 758.846,A -85,B 0,C 180,E1 -19941.915,E2 -19941.915} C_VEL
LIN {X 0,Y 227.892,Z 758.911,A -85,B 0,C 180,E1 -19946.373,E2 -19946.373} C_VEL
LIN {X 0,Y 227.905,Z 758.884,A -85,B 0,C 180,E1 -19950.436,E2 -19950.436} C_VEL
LIN {X 0,Y 227.93,Z 758.906,A -85,B 0,C 180,E1 -19954.426,E2 -19954.426} C_VEL
LIN {X 0,Y 227.963,Z 758.871,A -85,B 0,C 180,E1 -19958.287,E2 -19958.287} C_VEL
LIN {X 0,Y 228.036,Z 758.891,A -85,B 0,C 180,E1 -19962.826,E2 -19962.826} C_VEL
LIN {X 0,Y 228.076,Z 758.852,A -85,B 0,C 180,E1 -19967.544,E2 -19967.544} C_VEL
LIN {X 0,Y 228.301,Z 758.856,A -85,B 0,C 180,E1 -19971.146,E2 -19971.146} C_VEL
LIN {X 0,Y 228.351,Z 758.852,A -85,B 0,C 180,E1 -19972.929,E2 -19972.929} C_VEL
LIN {X 0,Y 228.556,Z 758.79,A -85,B 0,C 180,E1 -19978.238,E2 -19978.238} C_VEL
LIN {X 0,Y 228.559,Z 758.824,A -85,B 0,C 180,E1 -19981.762,E2 -19981.762} C_VEL
LIN {X 0,Y 228.357,Z 758.815,A -85,B 0,C 180,E1 -19987.072,E2 -19987.072} C_VEL
LIN {X 0,Y 228.16,Z 758.867,A -85,B 0,C 180,E1 -19990.651,E2 -19990.651} C_VEL
LIN {X 0,Y 228.048,Z 758.883,A -85,B 0,C 180,E1 -19994.273,E2 -19994.273} C_VEL
LIN {X 0,Y 227.957,Z 758.872,A -85,B 0,C 180,E1 -19997.957,E2 -19997.957} C_VEL
LIN {X 0,Y 227.917,Z 758.907,A -85,B 0,C 180,E1 -20002.32,E2 -20002.32} C_VEL
LIN {X 0,Y 227.943,Z 758.877,A -85,B 0,C 180,E1 -20006.602,E2 -20006.602} C_VEL
LIN {X 0,Y 227.898,Z 758.909,A -85,B 0,C 180,E1 -20010.291,E2 -20010.291} C_VEL
LIN {X 0,Y 227.879,Z 758.891,A -85,B 0,C 180,E1 -20013.72,E2 -20013.72} C_VEL
LIN {X 0,Y 227.845,Z 758.912,A -85,B 0,C 180,E1 -20018.091,E2 -20018.091} C_VEL
LIN {X 0,Y 227.805,Z 758.855,A -85,B 0,C 180,E1 -20022.744,E2 -20022.744} C_VEL
LIN {X 0,Y 227.811,Z 758.921,A -85,B 0,C 180,E1 -20027.258,E2 -20027.258} C_VEL
LIN {X 0,Y 227.845,Z 758.879,A -85,B 0,C 180,E1 -20031.909,E2 -20031.909} C_VEL
LIN {X 0,Y 227.88,Z 758.904,A -85,B 0,C 180,E1 -20036.378,E2 -20036.378} C_VEL
LIN {X 0,Y 227.901,Z 759.018,A -85,B 0,C 180,E1 -20041.193,E2 -20041.193} C_VEL
LIN {X 0,Y 228.119,Z 759.976,A -85,B 0,C 180,E1 -20041.693,E2 -20041.693} C_VEL
LIN {X 0,Y 229.185,Z 762.672,A -85,B 0,C 180,E1 -20042.046,E2 -20042.046} C_VEL
LIN {X 0,Y 235.167,Z 776.332,A -85,B 0,C 180,E1 -20043.284,E2 -20043.284} C_VEL
LIN {X 0,Y 239.329,Z 787.633,A -85,B 0,C 180,E1 -20044.16,E2 -20044.16} C_VEL
LIN {X 0,Y 240.466,Z 794.911,A -85,B 0,C 180,E1 -20044.529,E2 -20044.529} C_VEL
LIN {X 0,Y 239.168,Z 835.512,A -85,B 0,C 180,E1 -20045.749,E2 -20045.749} C_VEL
LIN {X 0,Y 238.704,Z 844.678,A -85,B 0,C 180,E1 -20046.231,E2 -20046.231} C_VEL
LIN {X 0,Y 237.822,Z 853.839,A -85,B 0,C 180,E1 -20046.913,E2 -20046.913} C_VEL
LIN {X 0,Y 236.706,Z 862.317,A -85,B 0,C 180,E1 -20047.756,E2 -20047.756} C_VEL
LIN {X 0,Y 235.471,Z 871.862,A -85,B 0,C 180,E1 -20049.013,E2 -20049.013} C_VEL
LIN {X 0,Y 233.627,Z 881.615,A -85,B 0,C 180,E1 -20050.676,E2 -20050.676} C_VEL
LIN {X 0,Y 232.124,Z 889.324,A -85,B 0,C 180,E1 -20052.376,E2 -20052.376} C_VEL
LIN {X 0,Y 230.726,Z 895.662,A -85,B 0,C 180,E1 -20054.089,E2 -20054.089} C_VEL
LIN {X 0,Y 229.544,Z 900.928,A -85,B 0,C 180,E1 -20055.822,E2 -20055.822} C_VEL
LIN {X 0,Y 228.487,Z 905.324,A -85,B 0,C 180,E1 -20057.566,E2 -20057.566} C_VEL
LIN {X 0,Y 227.337,Z 910.49,A -85,B 0,C 180,E1 -20060.21,E2 -20060.21} C_VEL
LIN {X 0,Y 226.742,Z 913.139,A -85,B 0,C 180,E1 -20061.982,E2 -20061.982} C_VEL
LIN {X 0,Y 226.381,Z 914.938,A -85,B 0,C 180,E1 -20063.435,E2 -20063.435} C_VEL
LIN {X 0,Y 225.927,Z 917.3,A -85,B 0,C 180,E1 -20066.433,E2 -20066.433} C_VEL
LIN {X 0,Y 225.779,Z 918.096,A -85,B 0,C 180,E1 -20068.216,E2 -20068.216} C_VEL
LIN {X 0,Y 225.748,Z 918.399,A -85,B 0,C 180,E1 -20070,E2 -20070} C_VEL
LIN {X 0,Y 225.777,Z 918.119,A -85,B 0,C 180,E1 -20071.784,E2 -20071.784} C_VEL
LIN {X 0,Y 225.922,Z 917.37,A -85,B 0,C 180,E1 -20073.567,E2 -20073.567} C_VEL
LIN {X 0,Y 226.378,Z 915.066,A -85,B 0,C 180,E1 -20076.557,E2 -20076.557} C_VEL
LIN {X 0,Y 226.995,Z 912.155,A -85,B 0,C 180,E1 -20078.906,E2 -20078.906} C_VEL
LIN {X 0,Y 227.985,Z 907.505,A -85,B 0,C 180,E1 -20081.559,E2 -20081.559} C_VEL
LIN {X 0,Y 229.216,Z 902.438,A -85,B 0,C 180,E1 -20083.746,E2 -20083.746} C_VEL
LIN {X 0,Y 230.376,Z 897.485,A -85,B 0,C 180,E1 -20085.482,E2 -20085.482} C_VEL
LIN {X 0,Y 231.741,Z 891.505,A -85,B 0,C 180,E1 -20087.199,E2 -20087.199} C_VEL
LIN {X 0,Y 233.146,Z 884.23,A -85,B 0,C 180,E1 -20088.908,E2 -20088.908} C_VEL
LIN {X 0,Y 234.658,Z 876.445,A -85,B 0,C 180,E1 -20090.375,E2 -20090.375} C_VEL
LIN {X 0,Y 236.045,Z 868.228,A -85,B 0,C 180,E1 -20091.62,E2 -20091.62} C_VEL
LIN {X 0,Y 237.44,Z 858.107,A -85,B 0,C 180,E1 -20092.819,E2 -20092.819} C_VEL
LIN {X 0,Y 238.612,Z 846.415,A -85,B 0,C 180,E1 -20093.79,E2 -20093.79} C_VEL
LIN {X 0,Y 239.185,Z 836.257,A -85,B 0,C 180,E1 -20094.347,E2 -20094.347} C_VEL
LIN {X 0,Y 240.424,Z 793.392,A -85,B 0,C 180,E1 -20095.658,E2 -20095.658} C_VEL
LIN {X 0,Y 239.06,Z 786.598,A -85,B 0,C 180,E1 -20096.039,E2 -20096.039} C_VEL
LIN {X 0,Y 233.119,Z 771.309,A -85,B 0,C 180,E1 -20097.279,E2 -20097.279} C_VEL
LIN {X 0,Y 228.248,Z 760.292,A -85,B 0,C 180,E1 -20098.366,E2 -20098.366} C_VEL
LIN {X 0,Y 227.933,Z 759.045,A -85,B 0,C 180,E1 -20098.913,E2 -20098.913} C_VEL
LIN {X 0,Y 227.878,Z 758.903,A -85,B 0,C 180,E1 -20103.72,E2 -20103.72} C_VEL
LIN {X 0,Y 227.845,Z 758.88,A -85,B 0,C 180,E1 -20108.091,E2 -20108.091} C_VEL
LIN {X 0,Y 227.811,Z 758.922,A -85,B 0,C 180,E1 -20112.742,E2 -20112.742} C_VEL
LIN {X 0,Y 227.805,Z 758.855,A -85,B 0,C 180,E1 -20117.256,E2 -20117.256} C_VEL
LIN {X 0,Y 227.845,Z 758.911,A -85,B 0,C 180,E1 -20121.909,E2 -20121.909} C_VEL
LIN {X 0,Y 227.881,Z 758.891,A -85,B 0,C 180,E1 -20126.377,E2 -20126.377} C_VEL
LIN {X 0,Y 227.905,Z 758.909,A -85,B 0,C 180,E1 -20130.436,E2 -20130.436} C_VEL
LIN {X 0,Y 227.926,Z 758.878,A -85,B 0,C 180,E1 -20134.425,E2 -20134.425} C_VEL
LIN {X 0,Y 227.949,Z 758.902,A -85,B 0,C 180,E1 -20138.286,E2 -20138.286} C_VEL
LIN {X 0,Y 228.006,Z 758.864,A -85,B 0,C 180,E1 -20142.851,E2 -20142.851} C_VEL
LIN {X 0,Y 228.071,Z 758.889,A -85,B 0,C 180,E1 -20147.543,E2 -20147.543} C_VEL
LIN {X 0,Y 228.327,Z 758.825,A -85,B 0,C 180,E1 -20151.147,E2 -20151.147} C_VEL
LIN {X 0,Y 228.36,Z 758.814,A -85,B 0,C 180,E1 -20152.929,E2 -20152.929} C_VEL
LIN {X 0,Y 228.559,Z 758.824,A -85,B 0,C 180,E1 -20158.238,E2 -20158.238} C_VEL
LIN {X 0,Y 228.556,Z 758.79,A -85,B 0,C 180,E1 -20161.762,E2 -20161.762} C_VEL
LIN {X 0,Y 228.351,Z 758.852,A -85,B 0,C 180,E1 -20167.071,E2 -20167.071} C_VEL
LIN {X 0,Y 228.16,Z 758.853,A -85,B 0,C 180,E1 -20170.65,E2 -20170.65} C_VEL
LIN {X 0,Y 228.066,Z 758.869,A -85,B 0,C 180,E1 -20174.272,E2 -20174.272} C_VEL
LIN {X 0,Y 228.005,Z 758.893,A -85,B 0,C 180,E1 -20177.953,E2 -20177.953} C_VEL
LIN {X 0,Y 227.931,Z 758.879,A -85,B 0,C 180,E1 -20182.329,E2 -20182.329} C_VEL
LIN {X 0,Y 227.943,Z 758.9,A -85,B 0,C 180,E1 -20186.602,E2 -20186.602} C_VEL
LIN {X 0,Y 227.865,Z 758.901,A -85,B 0,C 180,E1 -20191.213,E2 -20191.213} C_VEL
LIN {X 0,Y 227.902,Z 758.884,A -85,B 0,C 180,E1 -20195.868,E2 -20195.868} C_VEL
LIN {X 0,Y 227.845,Z 758.843,A -85,B 0,C 180,E1 -20198.87,E2 -20198.87} C_VEL
LIN {X 0,Y 227.168,Z 758.936,A -85,B 0,C 180,E1 -20200.345,E2 -20200.345} C_VEL
LIN {X 0,Y 224.283,Z 759.335,A -85,B 0,C 180,E1 -20202.751,E2 -20202.751} C_VEL
LIN {X 0,Y 221.848,Z 759.665,A -85,B 0,C 180,E1 -20204.714,E2 -20204.714} C_VEL
LIN {X 0,Y 220.828,Z 759.78,A -85,B 0,C 180,E1 -20206.24,E2 -20206.24} C_VEL
LIN {X 0,Y 220.758,Z 759.779,A -85,B 0,C 180,E1 -20206.757,E2 -20206.757} C_VEL
LIN {X 0,Y 220.809,Z 759.775,A -85,B 0,C 180,E1 -20210.464,E2 -20210.464} C_VEL
LIN {X 0,Y 220.888,Z 759.895,A -85,B 0,C 180,E1 -20214.922,E2 -20214.922} C_VEL
LIN {X 0,Y 222.399,Z 767.082,A -85,B 0,C 180,E1 -20218.879,E2 -20218.879} C_VEL
LIN {X 0,Y 223.264,Z 771.294,A -85,B 0,C 180,E1 -20220.949,E2 -20220.949} C_VEL
LIN {X 0,Y 225.555,Z 777.068,A -85,B 0,C 180,E1 -20221.553,E2 -20221.553} C_VEL
LIN {X 0,Y 228.931,Z 785.841,A -85,B 0,C 180,E1 -20222.31,E2 -20222.31} C_VEL
LIN {X 0,Y 232.249,Z 807.085,A -85,B 0,C 180,E1 -20223.456,E2 -20223.456} C_VEL
LIN {X 0,Y 233.446,Z 818.499,A -85,B 0,C 180,E1 -20223.984,E2 -20223.984} C_VEL
LIN {X 0,Y 232.387,Z 849.144,A -85,B 0,C 180,E1 -20224.951,E2 -20224.951} C_VEL
LIN {X 0,Y 231.436,Z 860.878,A -85,B 0,C 180,E1 -20225.607,E2 -20225.607} C_VEL
LIN {X 0,Y 230.065,Z 871.935,A -85,B 0,C 180,E1 -20226.602,E2 -20226.602} C_VEL
LIN {X 0,Y 228.768,Z 880.62,A -85,B 0,C 180,E1 -20227.656,E2 -20227.656} C_VEL
LIN {X 0,Y 227.257,Z 888.919,A -85,B 0,C 180,E1 -20228.93,E2 -20228.93} C_VEL
LIN {X 0,Y 225.707,Z 896.779,A -85,B 0,C 180,E1 -20230.444,E2 -20230.444} C_VEL
LIN {X 0,Y 224.066,Z 904.13,A -85,B 0,C 180,E1 -20232.193,E2 -20232.193} C_VEL
LIN {X 0,Y 222.299,Z 911.59,A -85,B 0,C 180,E1 -20234.411,E2 -20234.411} C_VEL
LIN {X 0,Y 220.944,Z 917.442,A -85,B 0,C 180,E1 -20236.667,E2 -20236.667} C_VEL
LIN {X 0,Y 219.934,Z 922.059,A -85,B 0,C 180,E1 -20238.946,E2 -20238.946} C_VEL
LIN {X 0,Y 219.335,Z 925.061,A -85,B 0,C 180,E1 -20240.781,E2 -20240.781} C_VEL
LIN {X 0,Y 218.943,Z 927.394,A -85,B 0,C 180,E1 -20242.623,E2 -20242.623} C_VEL
LIN {X 0,Y 218.582,Z 929.888,A -85,B 0,C 180,E1 -20245.366,E2 -20245.366} C_VEL
LIN {X 0,Y 218.57,Z 931.179,A -85,B 0,C 180,E1 -20248.157,E2 -20248.157} C_VEL
LIN {X 0,Y 218.631,Z 931.475,A -85,B 0,C 180,E1 -20250,E2 -20250} C_VEL
LIN {X 0,Y 218.57,Z 931.172,A -85,B 0,C 180,E1 -20251.843,E2 -20251.843} C_VEL
LIN {X 0,Y 218.565,Z 929.896,A -85,B 0,C 180,E1 -20254.579,E2 -20254.579} C_VEL
LIN {X 0,Y 218.944,Z 927.341,A -85,B 0,C 180,E1 -20257.377,E2 -20257.377} C_VEL
LIN {X 0,Y 219.607,Z 923.517,A -85,B 0,C 180,E1 -20260.138,E2 -20260.138} C_VEL
LIN {X 0,Y 220.705,Z 918.314,A -85,B 0,C 180,E1 -20262.88,E2 -20262.88} C_VEL
LIN {X 0,Y 222.298,Z 911.46,A -85,B 0,C 180,E1 -20265.589,E2 -20265.589} C_VEL
LIN {X 0,Y 224.057,Z 903.977,A -85,B 0,C 180,E1 -20267.808,E2 -20267.808} C_VEL
LIN {X 0,Y 225.673,Z 896.598,A -85,B 0,C 180,E1 -20269.559,E2 -20269.559} C_VEL
LIN {X 0,Y 227.246,Z 888.696,A -85,B 0,C 180,E1 -20271.071,E2 -20271.071} C_VEL
LIN {X 0,Y 228.759,Z 880.345,A -85,B 0,C 180,E1 -20272.345,E2 -20272.345} C_VEL
LIN {X 0,Y 230.231,Z 870.149,A -85,B 0,C 180,E1 -20273.562,E2 -20273.562} C_VEL
LIN {X 0,Y 231.556,Z 858.75,A -85,B 0,C 180,E1 -20274.493,E2 -20274.493} C_VEL
LIN {X 0,Y 232.301,Z 849.468,A -85,B 0,C 180,E1 -20275,E2 -20275} C_VEL
LIN {X 0,Y 233.253,Z 821.043,A -85,B 0,C 180,E1 -20275.909,E2 -20275.909} C_VEL
LIN {X 0,Y 233.21,Z 815.24,A -85,B 0,C 180,E1 -20276.108,E2 -20276.108} C_VEL
LIN {X 0,Y 229.713,Z 790.665,A -85,B 0,C 180,E1 -20277.375,E2 -20277.375} C_VEL
LIN {X 0,Y 228.535,Z 784.566,A -85,B 0,C 180,E1 -20277.738,E2 -20277.738} C_VEL
LIN {X 0,Y 223.296,Z 771.404,A -85,B 0,C 180,E1 -20278.975,E2 -20278.975} C_VEL
LIN {X 0,Y 222.288,Z 766.484,A -85,B 0,C 180,E1 -20281.39,E2 -20281.39} C_VEL
LIN {X 0,Y 220.885,Z 759.872,A -85,B 0,C 180,E1 -20285.079,E2 -20285.079} C_VEL
LIN {X 0,Y 220.809,Z 759.774,A -85,B 0,C 180,E1 -20289.536,E2 -20289.536} C_VEL
LIN {X 0,Y 220.776,Z 759.796,A -85,B 0,C 180,E1 -20294.454,E2 -20294.454} C_VEL
LIN {X 0,Y 220.789,Z 759.746,A -85,B 0,C 180,E1 -20298.052,E2 -20298.052} C_VEL
LIN {X 0,Y 220.834,Z 759.734,A -85,B 0,C 180,E1 -20302.795,E2 -20302.795} C_VEL
LIN {X 0,Y 220.824,Z 759.792,A -85,B 0,C 180,E1 -20307.245,E2 -20307.245} C_VEL
LIN {X 0,Y 220.828,Z 759.769,A -85,B 0,C 180,E1 -20311.485,E2 -20311.485} C_VEL
LIN {X 0,Y 220.869,Z 759.781,A -85,B 0,C 180,E1 -20315.565,E2 -20315.565} C_VEL
LIN {X 0,Y 220.894,Z 759.754,A -85,B 0,C 180,E1 -20319.514,E2 -20319.514} C_VEL
LIN {X 0,Y 221.018,Z 759.765,A -85,B 0,C 180,E1 -20323.371,E2 -20323.371} C_VEL
LIN {X 0,Y 221.108,Z 759.726,A -85,B 0,C 180,E1 -20329.006,E2 -20329.006} C_VEL
LIN {X 0,Y 221.286,Z 759.733,A -85,B 0,C 180,E1 -20332.702,E2 -20332.702} C_VEL
LIN {X 0,Y 221.514,Z 759.666,A -85,B 0,C 180,E1 -20338.182,E2 -20338.182} C_VEL
LIN {X 0,Y 221.517,Z 759.701,A -85,B 0,C 180,E1 -20341.818,E2 -20341.818} C_VEL
LIN {X 0,Y 221.292,Z 759.693,A -85,B 0,C 180,E1 -20347.299,E2 -20347.299} C_VEL
LIN {X 0,Y 221.107,Z 759.749,A -85,B 0,C 180,E1 -20350.995,E2 -20350.995} C_VEL
LIN {X 0,Y 220.981,Z 759.739,A -85,B 0,C 180,E1 -20356.633,E2 -20356.633} C_VEL
LIN {X 0,Y 220.879,Z 759.779,A -85,B 0,C 180,E1 -20360.488,E2 -20360.488} C_VEL
LIN {X 0,Y 220.863,Z 759.765,A -85,B 0,C 180,E1 -20364.436,E2 -20364.436} C_VEL
LIN {X 0,Y 220.828,Z 759.785,A -85,B 0,C 180,E1 -20368.515,E2 -20368.515} C_VEL
LIN {X 0,Y 220.818,Z 759.771,A -85,B 0,C 180,E1 -20372.756,E2 -20372.756} C_VEL
LIN {X 0,Y 220.813,Z 759.792,A -85,B 0,C 180,E1 -20377.279,E2 -20377.279} C_VEL
LIN {X 0,Y 220.765,Z 759.732,A -85,B 0,C 180,E1 -20381.954,E2 -20381.954} C_VEL
LIN {X 0,Y 220.772,Z 759.768,A -85,B 0,C 180,E1 -20385.545,E2 -20385.545} C_VEL
LIN {X 0,Y 220.808,Z 759.76,A -85,B 0,C 180,E1 -20390.463,E2 -20390.463} C_VEL
LIN {X 0,Y 220.802,Z 759.798,A -85,B 0,C 180,E1 -20395.045,E2 -20395.045} C_VEL
LIN {X 0,Y 220.835,Z 759.771,A -85,B 0,C 180,E1 -20399.39,E2 -20399.39} C_VEL
LIN {X 0,Y 220.877,Z 760.067,A -85,B 0,C 180,E1 -20400.545,E2 -20400.545} C_VEL
LIN {X 0,Y 221.245,Z 761.426,A -85,B 0,C 180,E1 -20400.873,E2 -20400.873} C_VEL
LIN {X 0,Y 226.887,Z 773.481,A -85,B 0,C 180,E1 -20402.115,E2 -20402.115} C_VEL
LIN {X 0,Y 233.048,Z 789.415,A -85,B 0,C 180,E1 -20403.462,E2 -20403.462} C_VEL
LIN {X 0,Y 234.092,Z 795.076,A -85,B 0,C 180,E1 -20403.781,E2 -20403.781} C_VEL
LIN {X 0,Y 232.73,Z 835.953,A -85,B 0,C 180,E1 -20405.043,E2 -20405.043} C_VEL
LIN {X 0,Y 232.193,Z 845.266,A -85,B 0,C 180,E1 -20405.548,E2 -20405.548} C_VEL
LIN {X 0,Y 231.169,Z 855.302,A -85,B 0,C 180,E1 -20406.331,E2 -20406.331} C_VEL
LIN {X 0,Y 229.795,Z 866.083,A -85,B 0,C 180,E1 -20407.524,E2 -20407.524} C_VEL
LIN {X 0,Y 228.084,Z 875.957,A -85,B 0,C 180,E1 -20409.01,E2 -20409.01} C_VEL
LIN {X 0,Y 226.55,Z 883.862,A -85,B 0,C 180,E1 -20410.52,E2 -20410.52} C_VEL
LIN {X 0,Y 225.041,Z 891.231,A -85,B 0,C 180,E1 -20412.272,E2 -20412.272} C_VEL
LIN {X 0,Y 223.276,Z 898.696,A -85,B 0,C 180,E1 -20414.481,E2 -20414.481} C_VEL
LIN {X 0,Y 221.575,Z 905.534,A -85,B 0,C 180,E1 -20417.172,E2 -20417.172} C_VEL
LIN {X 0,Y 220.35,Z 910.7,A -85,B 0,C 180,E1 -20419.897,E2 -20419.897} C_VEL
LIN {X 0,Y 219.729,Z 913.348,A -85,B 0,C 180,E1 -20421.725,E2 -20421.725} C_VEL
LIN {X 0,Y 219.073,Z 916.247,A -85,B 0,C 180,E1 -20424.477,E2 -20424.477} C_VEL
LIN {X 0,Y 218.84,Z 917.51,A -85,B 0,C 180,E1 -20426.317,E2 -20426.317} C_VEL
LIN {X 0,Y 218.699,Z 918.305,A -85,B 0,C 180,E1 -20428.158,E2 -20428.158} C_VEL
LIN {X 0,Y 218.663,Z 918.607,A -85,B 0,C 180,E1 -20430,E2 -20430} C_VEL
LIN {X 0,Y 218.697,Z 918.328,A -85,B 0,C 180,E1 -20431.842,E2 -20431.842} C_VEL
LIN {X 0,Y 218.835,Z 917.579,A -85,B 0,C 180,E1 -20433.683,E2 -20433.683} C_VEL
LIN {X 0,Y 219.253,Z 915.561,A -85,B 0,C 180,E1 -20436.441,E2 -20436.441} C_VEL
LIN {X 0,Y 219.972,Z 912.363,A -85,B 0,C 180,E1 -20439.192,E2 -20439.192} C_VEL
LIN {X 0,Y 221.04,Z 907.712,A -85,B 0,C 180,E1 -20441.927,E2 -20441.927} C_VEL
LIN {X 0,Y 222.314,Z 902.646,A -85,B 0,C 180,E1 -20444.182,E2 -20444.182} C_VEL
LIN {X 0,Y 223.549,Z 897.692,A -85,B 0,C 180,E1 -20445.967,E2 -20445.967} C_VEL
LIN {X 0,Y 224.979,Z 891.711,A -85,B 0,C 180,E1 -20447.733,E2 -20447.733} C_VEL
LIN {X 0,Y 226.461,Z 884.434,A -85,B 0,C 180,E1 -20449.488,E2 -20449.488} C_VEL
LIN {X 0,Y 228.027,Z 876.649,A -85,B 0,C 180,E1 -20450.995,E2 -20450.995} C_VEL
LIN {X 0,Y 229.482,Z 868.431,A -85,B 0,C 180,E1 -20452.271,E2 -20452.271} C_VEL
LIN {X 0,Y 230.922,Z 858.393,A -85,B 0,C 180,E1 -20453.491,E2 -20453.491} C_VEL
LIN {X 0,Y 232.16,Z 846.279,A -85,B 0,C 180,E1 -20454.518,E2 -20454.518} C_VEL
LIN {X 0,Y 232.746,Z 836.309,A -85,B 0,C 180,E1 -20455.073,E2 -20455.073} C_VEL
LIN {X 0,Y 234.069,Z 794.441,A -85,B 0,C 180,E1 -20456.378,E2 -20456.378} C_VEL
LIN {X 0,Y 232.847,Z 788.746,A -85,B 0,C 180,E1 -20456.722,E2 -20456.722} C_VEL
LIN {X 0,Y 227,Z 773.65,A -85,B 0,C 180,E1 -20458.003,E2 -20458.003} C_VEL
LIN {X 0,Y 221.667,Z 762.314,A -85,B 0,C 180,E1 -20459.156,E2 -20459.156} C_VEL
LIN {X 0,Y 220.948,Z 760.392,A -85,B 0,C 180,E1 -20459.458,E2 -20459.458} C_VEL
LIN {X 0,Y 220.843,Z 759.835,A -85,B 0,C 180,E1 -20459.927,E2 -20459.927} C_VEL
LIN {X 0,Y 220.809,Z 759.791,A -85,B 0,C 180,E1 -20464.153,E2 -20464.153} C_VEL
LIN {X 0,Y 220.811,Z 759.761,A -85,B 0,C 180,E1 -20467.278,E2 -20467.278} C_VEL
LIN {X 0,Y 220.796,Z 759.768,A -85,B 0,C 180,E1 -20470.188,E2 -20470.188} C_VEL
LIN {X 0,Y 220.772,Z 759.772,A -85,B 0,C 180,E1 -20474.455,E2 -20474.455} C_VEL
LIN {X 0,Y 220.765,Z 759.732,A -85,B 0,C 180,E1 -20478.046,E2 -20478.046} C_VEL
LIN {X 0,Y 220.826,Z 759.79,A -85,B 0,C 180,E1 -20482.793,E2 -20482.793} C_VEL
LIN {X 0,Y 220.818,Z 759.771,A -85,B 0,C 180,E1 -20487.244,E2 -20487.244} C_VEL
LIN {X 0,Y 220.828,Z 759.785,A -85,B 0,C 180,E1 -20491.485,E2 -20491.485} C_VEL
LIN {X 0,Y 220.863,Z 759.764,A -85,B 0,C 180,E1 -20495.564,E2 -20495.564} C_VEL
LIN {X 0,Y 220.883,Z 759.779,A -85,B 0,C 180,E1 -20499.513,E2 -20499.513} C_VEL
LIN {X 0,Y 220.988,Z 759.738,A -85,B 0,C 180,E1 -20503.368,E2 -20503.368} C_VEL
LIN {X 0,Y 221.112,Z 759.749,A -85,B 0,C 180,E1 -20509.006,E2 -20509.006} C_VEL
LIN {X 0,Y 221.297,Z 759.693,A -85,B 0,C 180,E1 -20512.702,E2 -20512.702} C_VEL
LIN {X 0,Y 221.517,Z 759.701,A -85,B 0,C 180,E1 -20518.182,E2 -20518.182} C_VEL
LIN {X 0,Y 221.514,Z 759.667,A -85,B 0,C 180,E1 -20521.818,E2 -20521.818} C_VEL
LIN {X 0,Y 221.286,Z 759.733,A -85,B 0,C 180,E1 -20527.298,E2 -20527.298} C_VEL
LIN {X 0,Y 221.108,Z 759.726,A -85,B 0,C 180,E1 -20530.994,E2 -20530.994} C_VEL
LIN {X 0,Y 221.018,Z 759.766,A -85,B 0,C 180,E1 -20536.629,E2 -20536.629} C_VEL
LIN {X 0,Y 220.894,Z 759.753,A -85,B 0,C 180,E1 -20540.486,E2 -20540.486} C_VEL
LIN {X 0,Y 220.869,Z 759.782,A -85,B 0,C 180,E1 -20544.435,E2 -20544.435} C_VEL
LIN {X 0,Y 220.828,Z 759.768,A -85,B 0,C 180,E1 -20548.515,E2 -20548.515} C_VEL
LIN {X 0,Y 220.824,Z 759.792,A -85,B 0,C 180,E1 -20552.755,E2 -20552.755} C_VEL
LIN {X 0,Y 220.839,Z 759.73,A -85,B 0,C 180,E1 -20557.288,E2 -20557.288} C_VEL
LIN {X 0,Y 220.789,Z 759.749,A -85,B 0,C 180,E1 -20561.948,E2 -20561.948} C_VEL
LIN {X 0,Y 220.776,Z 759.795,A -85,B 0,C 180,E1 -20565.546,E2 -20565.546} C_VEL
LIN {X 0,Y 220.758,Z 759.779,A -85,B 0,C 180,E1 -20566.757,E2 -20566.757} C_VEL
LIN {X 0,Y 220.099,Z 759.856,A -85,B 0,C 180,E1 -20567.771,E2 -20567.771} C_VEL
LIN {X 0,Y 217.265,Z 760.215,A -85,B 0,C 180,E1 -20569.366,E2 -20569.366} C_VEL
LIN {X 0,Y 214.415,Z 760.583,A -85,B 0,C 180,E1 -20571,E2 -20571} C_VEL
LIN {X 0,Y 213.772,Z 760.668,A -85,B 0,C 180,E1 -20572.061,E2 -20572.061} C_VEL
LIN {X 0,Y 213.851,Z 760.833,A -85,B 0,C 180,E1 -20574.239,E2 -20574.239} C_VEL
LIN {X 0,Y 215.473,Z 768.354,A -85,B 0,C 180,E1 -20578.542,E2 -20578.542} C_VEL
LIN {X 0,Y 216.032,Z 771.154,A -85,B 0,C 180,E1 -20579.897,E2 -20579.897} C_VEL
LIN {X 0,Y 221.838,Z 785.225,A -85,B 0,C 180,E1 -20581.33,E2 -20581.33} C_VEL
LIN {X 0,Y 223.06,Z 789.305,A -85,B 0,C 180,E1 -20581.646,E2 -20581.646} C_VEL
LIN {X 0,Y 226.192,Z 810.083,A -85,B 0,C 180,E1 -20582.798,E2 -20582.798} C_VEL
LIN {X 0,Y 227.071,Z 818.564,A -85,B 0,C 180,E1 -20583.205,E2 -20583.205} C_VEL
LIN {X 0,Y 225.976,Z 848.951,A -85,B 0,C 180,E1 -20584.189,E2 -20584.189} C_VEL
LIN {X 0,Y 225.132,Z 859.238,A -85,B 0,C 180,E1 -20584.766,E2 -20584.766} C_VEL
LIN {X 0,Y 223.838,Z 870.028,A -85,B 0,C 180,E1 -20585.687,E2 -20585.687} C_VEL
LIN {X 0,Y 222.215,Z 880.416,A -85,B 0,C 180,E1 -20586.959,E2 -20586.959} C_VEL
LIN {X 0,Y 220.629,Z 888.713,A -85,B 0,C 180,E1 -20588.265,E2 -20588.265} C_VEL
LIN {X 0,Y 219.028,Z 896.573,A -85,B 0,C 180,E1 -20589.822,E2 -20589.822} C_VEL
LIN {X 0,Y 217.302,Z 903.924,A -85,B 0,C 180,E1 -20591.619,E2 -20591.619} C_VEL
LIN {X 0,Y 215.466,Z 911.383,A -85,B 0,C 180,E1 -20593.904,E2 -20593.904} C_VEL
LIN {X 0,Y 214.037,Z 917.234,A -85,B 0,C 180,E1 -20596.228,E2 -20596.228} C_VEL
LIN {X 0,Y 212.964,Z 921.851,A -85,B 0,C 180,E1 -20598.58,E2 -20598.58} C_VEL
LIN {X 0,Y 212.307,Z 924.853,A -85,B 0,C 180,E1 -20600.473,E2 -20600.473} C_VEL
LIN {X 0,Y 211.883,Z 927.185,A -85,B 0,C 180,E1 -20602.376,E2 -20602.376} C_VEL
LIN {X 0,Y 211.506,Z 929.813,A -85,B 0,C 180,E1 -20605.451,E2 -20605.451} C_VEL
LIN {X 0,Y 211.471,Z 930.97,A -85,B 0,C 180,E1 -20608.095,E2 -20608.095} C_VEL
LIN {X 0,Y 211.548,Z 931.267,A -85,B 0,C 180,E1 -20610,E2 -20610} C_VEL
LIN {X 0,Y 211.47,Z 930.963,A -85,B 0,C 180,E1 -20611.905,E2 -20611.905} C_VEL
LIN {X 0,Y 211.472,Z 929.848,A -85,B 0,C 180,E1 -20614.434,E2 -20614.434} C_VEL
LIN {X 0,Y 211.884,Z 927.131,A -85,B 0,C 180,E1 -20617.624,E2 -20617.624} C_VEL
LIN {X 0,Y 212.616,Z 923.307,A -85,B 0,C 180,E1 -20620.475,E2 -20620.475} C_VEL
LIN {X 0,Y 213.779,Z 918.103,A -85,B 0,C 180,E1 -20623.305,E2 -20623.305} C_VEL
LIN {X 0,Y 215.465,Z 911.249,A -85,B 0,C 180,E1 -20626.096,E2 -20626.096} C_VEL
LIN {X 0,Y 217.293,Z 903.765,A -85,B 0,C 180,E1 -20628.382,E2 -20628.382} C_VEL
LIN {X 0,Y 218.993,Z 896.386,A -85,B 0,C 180,E1 -20630.181,E2 -20630.181} C_VEL
LIN {X 0,Y 220.637,Z 888.483,A -85,B 0,C 180,E1 -20631.734,E2 -20631.734} C_VEL
LIN {X 0,Y 222.216,Z 880.132,A -85,B 0,C 180,E1 -20633.041,E2 -20633.041} C_VEL
LIN {X 0,Y 223.839,Z 869.235,A -85,B 0,C 180,E1 -20634.361,E2 -20634.361} C_VEL
LIN {X 0,Y 225.195,Z 857.79,A -85,B 0,C 180,E1 -20635.287,E2 -20635.287} C_VEL
LIN {X 0,Y 225.954,Z 847.957,A -85,B 0,C 180,E1 -20635.814,E2 -20635.814} C_VEL
LIN {X 0,Y 226.92,Z 816.785,A -85,B 0,C 180,E1 -20636.828,E2 -20636.828} C_VEL
LIN {X 0,Y 223.469,Z 792.098,A -85,B 0,C 180,E1 -20638.148,E2 -20638.148} C_VEL
LIN {X 0,Y 222.468,Z 787.01,A -85,B 0,C 180,E1 -20638.467,E2 -20638.467} C_VEL
LIN {X 0,Y 217.02,Z 773.755,A -85,B 0,C 180,E1 -20639.735,E2 -20639.735} C_VEL
LIN {X 0,Y 215.985,Z 770.999,A -85,B 0,C 180,E1 -20640.09,E2 -20640.09} C_VEL
LIN {X 0,Y 214.542,Z 764.012,A -85,B 0,C 180,E1 -20643.841,E2 -20643.841} C_VEL
LIN {X 0,Y 213.844,Z 760.699,A -85,B 0,C 180,E1 -20645.861,E2 -20645.861} C_VEL
LIN {X 0,Y 213.721,Z 760.644,A -85,B 0,C 180,E1 -20650.858,E2 -20650.858} C_VEL
LIN {X 0,Y 213.708,Z 760.667,A -85,B 0,C 180,E1 -20653.678,E2 -20653.678} C_VEL
LIN {X 0,Y 213.748,Z 760.662,A -85,B 0,C 180,E1 -20656.332,E2 -20656.332} C_VEL
LIN {X 0,Y 213.737,Z 760.599,A -85,B 0,C 180,E1 -20661.336,E2 -20661.336} C_VEL
LIN {X 0,Y 213.771,Z 760.668,A -85,B 0,C 180,E1 -20666.021,E2 -20666.021} C_VEL
LIN {X 0,Y 213.761,Z 760.645,A -85,B 0,C 180,E1 -20670.451,E2 -20670.451} C_VEL
LIN {X 0,Y 213.803,Z 760.664,A -85,B 0,C 180,E1 -20674.702,E2 -20674.702} C_VEL
LIN {X 0,Y 213.814,Z 760.632,A -85,B 0,C 180,E1 -20678.804,E2 -20678.804} C_VEL
LIN {X 0,Y 213.945,Z 760.647,A -85,B 0,C 180,E1 -20682.804,E2 -20682.804} C_VEL
LIN {X 0,Y 213.956,Z 760.614,A -85,B 0,C 180,E1 -20686.707,E2 -20686.707} C_VEL
LIN {X 0,Y 214.165,Z 760.609,A -85,B 0,C 180,E1 -20690.556,E2 -20690.556} C_VEL
LIN {X 0,Y 214.224,Z 760.615,A -85,B 0,C 180,E1 -20692.46,E2 -20692.46} C_VEL
LIN {X 0,Y 214.447,Z 760.546,A -85,B 0,C 180,E1 -20698.122,E2 -20698.122} C_VEL
LIN {X 0,Y 214.552,Z 760.554,A -85,B 0,C 180,E1 -20700,E2 -20700} C_VEL
LIN {X 0,Y 214.45,Z 760.581,A -85,B 0,C 180,E1 -20701.878,E2 -20701.878} C_VEL
LIN {X 0,Y 214.23,Z 760.572,A -85,B 0,C 180,E1 -20707.541,E2 -20707.541} C_VEL
LIN {X 0,Y 214.023,Z 760.635,A -85,B 0,C 180,E1 -20711.363,E2 -20711.363} C_VEL
LIN {X 0,Y 213.909,Z 760.634,A -85,B 0,C 180,E1 -20715.239,E2 -20715.239} C_VEL
LIN {X 0,Y 213.817,Z 760.644,A -85,B 0,C 180,E1 -20719.19,E2 -20719.19} C_VEL
LIN {X 0,Y 213.812,Z 760.657,A -85,B 0,C 180,E1 -20723.231,E2 -20723.231} C_VEL
LIN {X 0,Y 213.831,Z 760.642,A -85,B 0,C 180,E1 -20727.45,E2 -20727.45} C_VEL
LIN {X 0,Y 213.769,Z 760.659,A -85,B 0,C 180,E1 -20731.738,E2 -20731.738} C_VEL
LIN {X 0,Y 213.745,Z 760.672,A -85,B 0,C 180,E1 -20736.288,E2 -20736.288} C_VEL
LIN {X 0,Y 213.709,Z 760.616,A -85,B 0,C 180,E1 -20741.126,E2 -20741.126} C_VEL
LIN {X 0,Y 213.704,Z 760.614,A -85,B 0,C 180,E1 -20743.679,E2 -20743.679} C_VEL
LIN {X 0,Y 213.705,Z 760.666,A -85,B 0,C 180,E1 -20746.345,E2 -20746.345} C_VEL
LIN {X 0,Y 213.718,Z 760.662,A -85,B 0,C 180,E1 -20749.143,E2 -20749.143} C_VEL
LIN {X 0,Y 213.745,Z 760.651,A -85,B 0,C 180,E1 -20753.712,E2 -20753.712} C_VEL
LIN {X 0,Y 213.76,Z 760.646,A -85,B 0,C 180,E1 -20758.261,E2 -20758.261} C_VEL
LIN {X 0,Y 213.842,Z 760.932,A -85,B 0,C 180,E1 -20759.51,E2 -20759.51} C_VEL
LIN {X 0,Y 214.179,Z 762.234,A -85,B 0,C 180,E1 -20759.838,E2 -20759.838} C_VEL
LIN {X 0,Y 218.715,Z 771.244,A -85,B 0,C 180,E1 -20760.883,E2 -20760.883} C_VEL
LIN {X 0,Y 224.633,Z 785.406,A -85,B 0,C 180,E1 -20762.232,E2 -20762.232} C_VEL
LIN {X 0,Y 227.144,Z 792.585,A -85,B 0,C 180,E1 -20762.819,E2 -20762.819} C_VEL
LIN {X 0,Y 227.708,Z 796.417,A -85,B 0,C 180,E1 -20763.025,E2 -20763.025} C_VEL
LIN {X 0,Y 226.333,Z 836.179,A -85,B 0,C 180,E1 -20764.287,E2 -20764.287} C_VEL
LIN {X 0,Y 225.776,Z 845.358,A -85,B 0,C 180,E1 -20764.795,E2 -20764.795} C_VEL
LIN {X 0,Y 224.678,Z 855.72,A -85,B 0,C 180,E1 -20765.624,E2 -20765.624} C_VEL
LIN {X 0,Y 223.263,Z 866.297,A -85,B 0,C 180,E1 -20766.829,E2 -20766.829} C_VEL
LIN {X 0,Y 221.485,Z 876.17,A -85,B 0,C 180,E1 -20768.354,E2 -20768.354} C_VEL
LIN {X 0,Y 219.887,Z 884.074,A -85,B 0,C 180,E1 -20769.904,E2 -20769.904} C_VEL
LIN {X 0,Y 218.299,Z 891.442,A -85,B 0,C 180,E1 -20771.706,E2 -20771.706} C_VEL
LIN {X 0,Y 216.46,Z 898.907,A -85,B 0,C 180,E1 -20773.98,E2 -20773.98} C_VEL
LIN {X 0,Y 214.677,Z 905.744,A -85,B 0,C 180,E1 -20776.752,E2 -20776.752} C_VEL
LIN {X 0,Y 213.368,Z 910.91,A -85,B 0,C 180,E1 -20779.563,E2 -20779.563} C_VEL
LIN {X 0,Y 212.716,Z 913.558,A -85,B 0,C 180,E1 -20781.45,E2 -20781.45} C_VEL
LIN {X 0,Y 212.02,Z 916.457,A -85,B 0,C 180,E1 -20784.293,E2 -20784.293} C_VEL
LIN {X 0,Y 211.756,Z 917.719,A -85,B 0,C 180,E1 -20786.194,E2 -20786.194} C_VEL
LIN {X 0,Y 211.621,Z 918.513,A -85,B 0,C 180,E1 -20788.097,E2 -20788.097} C_VEL
LIN {X 0,Y 211.581,Z 918.816,A -85,B 0,C 180,E1 -20790,E2 -20790} C_VEL
LIN {X 0,Y 211.619,Z 918.536,A -85,B 0,C 180,E1 -20791.903,E2 -20791.903} C_VEL
LIN {X 0,Y 211.751,Z 917.787,A -85,B 0,C 180,E1 -20793.806,E2 -20793.806} C_VEL
LIN {X 0,Y 212.133,Z 916.047,A -85,B 0,C 180,E1 -20796.327,E2 -20796.327} C_VEL
LIN {X 0,Y 212.667,Z 913.721,A -85,B 0,C 180,E1 -20798.552,E2 -20798.552} C_VEL
LIN {X 0,Y 213.296,Z 911.125,A -85,B 0,C 180,E1 -20800.441,E2 -20800.441} C_VEL
LIN {X 0,Y 214.594,Z 906.017,A -85,B 0,C 180,E1 -20803.253,E2 -20803.253} C_VEL
LIN {X 0,Y 216.074,Z 900.516,A -85,B 0,C 180,E1 -20805.565,E2 -20805.565} C_VEL
LIN {X 0,Y 217.875,Z 893.598,A -85,B 0,C 180,E1 -20807.845,E2 -20807.845} C_VEL
LIN {X 0,Y 219.588,Z 885.657,A -85,B 0,C 180,E1 -20809.88,E2 -20809.88} C_VEL
LIN {X 0,Y 221.176,Z 878.08,A -85,B 0,C 180,E1 -20811.433,E2 -20811.433} C_VEL
LIN {X 0,Y 222.68,Z 870.132,A -85,B 0,C 180,E1 -20812.745,E2 -20812.745} C_VEL
LIN {X 0,Y 223.98,Z 861.915,A -85,B 0,C 180,E1 -20813.828,E2 -20813.828} C_VEL
LIN {X 0,Y 225.048,Z 853.695,A -85,B 0,C 180,E1 -20814.676,E2 -20814.676} C_VEL
LIN {X 0,Y 225.887,Z 844.238,A -85,B 0,C 180,E1 -20815.412,E2 -20815.412} C_VEL
LIN {X 0,Y 226.48,Z 834.171,A -85,B 0,C 180,E1 -20815.928,E2 -20815.928} C_VEL
LIN {X 0,Y 227.74,Z 795.476,A -85,B 0,C 180,E1 -20817.141,E2 -20817.141} C_VEL
LIN {X 0,Y 226.611,Z 790.613,A -85,B 0,C 180,E1 -20817.459,E2 -20817.459} C_VEL
LIN {X 0,Y 220.496,Z 775.215,A -85,B 0,C 180,E1 -20818.855,E2 -20818.855} C_VEL
LIN {X 0,Y 215.376,Z 764.35,A -85,B 0,C 180,E1 -20820.024,E2 -20820.024} C_VEL
LIN {X 0,Y 213.989,Z 761.598,A -85,B 0,C 180,E1 -20820.405,E2 -20820.405} C_VEL
LIN {X 0,Y 213.795,Z 760.734,A -85,B 0,C 180,E1 -20820.822,E2 -20820.822} C_VEL
LIN {X 0,Y 213.773,Z 760.675,A -85,B 0,C 180,E1 -20824.724,E2 -20824.724} C_VEL
LIN {X 0,Y 213.723,Z 760.636,A -85,B 0,C 180,E1 -20828.667,E2 -20828.667} C_VEL
LIN {X 0,Y 213.713,Z 760.665,A -85,B 0,C 180,E1 -20831.125,E2 -20831.125} C_VEL
LIN {X 0,Y 213.706,Z 760.668,A -85,B 0,C 180,E1 -20833.679,E2 -20833.679} C_VEL
LIN {X 0,Y 213.704,Z 760.616,A -85,B 0,C 180,E1 -20836.345,E2 -20836.345} C_VEL
LIN {X 0,Y 213.715,Z 760.617,A -85,B 0,C 180,E1 -20839.144,E2 -20839.144} C_VEL
LIN {X 0,Y 213.745,Z 760.672,A -85,B 0,C 180,E1 -20843.712,E2 -20843.712} C_VEL
LIN {X 0,Y 213.769,Z 760.657,A -85,B 0,C 180,E1 -20848.262,E2 -20848.262} C_VEL
LIN {X 0,Y 213.828,Z 760.643,A -85,B 0,C 180,E1 -20852.603,E2 -20852.603} C_VEL
LIN {X 0,Y 213.821,Z 760.656,A -85,B 0,C 180,E1 -20856.973,E2 -20856.973} C_VEL
LIN {X 0,Y 213.919,Z 760.617,A -85,B 0,C 180,E1 -20862.801,E2 -20862.801} C_VEL
LIN {X 0,Y 213.945,Z 760.645,A -85,B 0,C 180,E1 -20866.706,E2 -20866.706} C_VEL
LIN {X 0,Y 214.198,Z 760.591,A -85,B 0,C 180,E1 -20870.557,E2 -20870.557} C_VEL
LIN {X 0,Y 214.237,Z 760.571,A -85,B 0,C 180,E1 -20872.46,E2 -20872.46} C_VEL
LIN {X 0,Y 214.45,Z 760.581,A -85,B 0,C 180,E1 -20878.122,E2 -20878.122} C_VEL
LIN {X 0,Y 214.552,Z 760.555,A -85,B 0,C 180,E1 -20880,E2 -20880} C_VEL
LIN {X 0,Y 214.447,Z 760.546,A -85,B 0,C 180,E1 -20881.878,E2 -20881.878} C_VEL
LIN {X 0,Y 214.224,Z 760.614,A -85,B 0,C 180,E1 -20887.54,E2 -20887.54} C_VEL
LIN {X 0,Y 214.025,Z 760.604,A -85,B 0,C 180,E1 -20891.363,E2 -20891.363} C_VEL
LIN {X 0,Y 213.936,Z 760.641,A -85,B 0,C 180,E1 -20895.237,E2 -20895.237} C_VEL
LIN {X 0,Y 213.841,Z 760.645,A -85,B 0,C 180,E1 -20899.187,E2 -20899.187} C_VEL
LIN {X 0,Y 213.848,Z 760.643,A -85,B 0,C 180,E1 -20903.227,E2 -20903.227} C_VEL
LIN {X 0,Y 213.83,Z 760.65,A -85,B 0,C 180,E1 -20907.45,E2 -20907.45} C_VEL
LIN {X 0,Y 213.771,Z 760.663,A -85,B 0,C 180,E1 -20911.737,E2 -20911.737} C_VEL
LIN {X 0,Y 213.755,Z 760.631,A -85,B 0,C 180,E1 -20916.286,E2 -20916.286} C_VEL
LIN {X 0,Y 213.725,Z 760.612,A -85,B 0,C 180,E1 -20921.122,E2 -20921.122} C_VEL
LIN {X 0,Y 213.748,Z 760.663,A -85,B 0,C 180,E1 -20923.668,E2 -20923.668} C_VEL
LIN {X 0,Y 213.716,Z 760.644,A -85,B 0,C 180,E1 -20928.876,E2 -20928.876} C_VEL
LIN {X 0,Y 213.772,Z 760.668,A -85,B 0,C 180,E1 -20932.061,E2 -20932.061} C_VEL
LIN {X 0,Y 213.194,Z 761.12,A -85,B 0,C 180,E1 -20933.104,E2 -20933.104} C_VEL
LIN {X 0,Y 211.282,Z 762.719,A -85,B 0,C 180,E1 -20934.392,E2 -20934.392} C_VEL
LIN {X 0,Y 208.429,Z 766.225,A -85,B 0,C 180,E1 -20936.272,E2 -20936.272} C_VEL
LIN {X 0,Y 208.15,Z 768.058,A -85,B 0,C 180,E1 -20937.269,E2 -20937.269} C_VEL
LIN {X 0,Y 208.77,Z 770.893,A -85,B 0,C 180,E1 -20938.731,E2 -20938.731} C_VEL
LIN {X 0,Y 214.896,Z 785.399,A -85,B 0,C 180,E1 -20940.327,E2 -20940.327} C_VEL
LIN {X 0,Y 216.893,Z 790.907,A -85,B 0,C 180,E1 -20940.83,E2 -20940.83} C_VEL
LIN {X 0,Y 219.739,Z 810.04,A -85,B 0,C 180,E1 -20941.935,E2 -20941.935} C_VEL
LIN {X 0,Y 220.684,Z 818.515,A -85,B 0,C 180,E1 -20942.37,E2 -20942.37} C_VEL
LIN {X 0,Y 219.608,Z 848.758,A -85,B 0,C 180,E1 -20943.382,E2 -20943.382} C_VEL
LIN {X 0,Y 218.656,Z 859.883,A -85,B 0,C 180,E1 -20944.029,E2 -20944.029} C_VEL
LIN {X 0,Y 217.12,Z 871.529,A -85,B 0,C 180,E1 -20945.115,E2 -20945.115} C_VEL
LIN {X 0,Y 215.708,Z 880.212,A -85,B 0,C 180,E1 -20946.222,E2 -20946.222} C_VEL
LIN {X 0,Y 214.053,Z 888.508,A -85,B 0,C 180,E1 -20947.562,E2 -20947.562} C_VEL
LIN {X 0,Y 212.376,Z 896.368,A -85,B 0,C 180,E1 -20949.161,E2 -20949.161} C_VEL
LIN {X 0,Y 210.554,Z 903.717,A -85,B 0,C 180,E1 -20951.008,E2 -20951.008} C_VEL
LIN {X 0,Y 208.643,Z 911.175,A -85,B 0,C 180,E1 -20953.362,E2 -20953.362} C_VEL
LIN {X 0,Y 206.877,Z 917.988,A -85,B 0,C 180,E1 -20956.243,E2 -20956.243} C_VEL
LIN {X 0,Y 205.615,Z 923.169,A -85,B 0,C 180,E1 -20959.164,E2 -20959.164} C_VEL
LIN {X 0,Y 204.831,Z 926.977,A -85,B 0,C 180,E1 -20962.112,E2 -20962.112} C_VEL
LIN {X 0,Y 204.41,Z 929.762,A -85,B 0,C 180,E1 -20965.613,E2 -20965.613} C_VEL
LIN {X 0,Y 204.376,Z 930.761,A -85,B 0,C 180,E1 -20968.029,E2 -20968.029} C_VEL
LIN {X 0,Y 204.466,Z 931.058,A -85,B 0,C 180,E1 -20970,E2 -20970} C_VEL
LIN {X 0,Y 204.373,Z 930.753,A -85,B 0,C 180,E1 -20971.971,E2 -20971.971} C_VEL
LIN {X 0,Y 204.383,Z 929.787,A -85,B 0,C 180,E1 -20974.288,E2 -20974.288} C_VEL
LIN {X 0,Y 204.832,Z 926.921,A -85,B 0,C 180,E1 -20977.888,E2 -20977.888} C_VEL
LIN {X 0,Y 205.614,Z 923.096,A -85,B 0,C 180,E1 -20980.836,E2 -20980.836} C_VEL
LIN {X 0,Y 206.874,Z 917.893,A -85,B 0,C 180,E1 -20983.757,E2 -20983.757} C_VEL
LIN {X 0,Y 208.642,Z 911.037,A -85,B 0,C 180,E1 -20986.638,E2 -20986.638} C_VEL
LIN {X 0,Y 210.546,Z 903.553,A -85,B 0,C 180,E1 -20988.993,E2 -20988.993} C_VEL
LIN {X 0,Y 212.33,Z 896.174,A -85,B 0,C 180,E1 -20990.844,E2 -20990.844} C_VEL
LIN {X 0,Y 214.061,Z 888.271,A -85,B 0,C 180,E1 -20992.437,E2 -20992.437} C_VEL
LIN {X 0,Y 215.877,Z 878.886,A -85,B 0,C 180,E1 -20993.933,E2 -20993.933} C_VEL
LIN {X 0,Y 217.597,Z 867.378,A -85,B 0,C 180,E1 -20995.286,E2 -20995.286} C_VEL
LIN {X 0,Y 218.815,Z 857.571,A -85,B 0,C 180,E1 -20996.079,E2 -20996.079} C_VEL
LIN {X 0,Y 219.585,Z 847.732,A -85,B 0,C 180,E1 -20996.621,E2 -20996.621} C_VEL
LIN {X 0,Y 220.575,Z 817.467,A -85,B 0,C 180,E1 -20997.631,E2 -20997.631} C_VEL
LIN {X 0,Y 217.332,Z 793.968,A -85,B 0,C 180,E1 -20998.939,E2 -20998.939} C_VEL
LIN {X 0,Y 216.333,Z 789.155,A -85,B 0,C 180,E1 -20999.263,E2 -20999.263} C_VEL
LIN {X 0,Y 210.313,Z 774.531,A -85,B 0,C 180,E1 -21000.744,E2 -21000.744} C_VEL
LIN {X 0,Y 208.748,Z 770.836,A -85,B 0,C 180,E1 -21001.225,E2 -21001.225} C_VEL
LIN {X 0,Y 207.486,Z 764.837,A -85,B 0,C 180,E1 -21004.566,E2 -21004.566} C_VEL
LIN {X 0,Y 206.754,Z 761.568,A -85,B 0,C 180,E1 -21006.653,E2 -21006.653} C_VEL
LIN {X 0,Y 206.645,Z 761.524,A -85,B 0,C 180,E1 -21011.564,E2 -21011.564} C_VEL
LIN {X 0,Y 206.66,Z 761.553,A -85,B 0,C 180,E1 -21015.574,E2 -21015.574} C_VEL
LIN {X 0,Y 206.672,Z 761.478,A -85,B 0,C 180,E1 -21019.752,E2 -21019.752} C_VEL
LIN {X 0,Y 206.732,Z 761.528,A -85,B 0,C 180,E1 -21024.695,E2 -21024.695} C_VEL
LIN {X 0,Y 206.708,Z 761.528,A -85,B 0,C 180,E1 -21029.337,E2 -21029.337} C_VEL
LIN {X 0,Y 206.734,Z 761.545,A -85,B 0,C 180,E1 -21033.773,E2 -21033.773} C_VEL
LIN {X 0,Y 206.758,Z 761.512,A -85,B 0,C 180,E1 -21038.044,E2 -21038.044} C_VEL
LIN {X 0,Y 206.875,Z 761.526,A -85,B 0,C 180,E1 -21042.197,E2 -21042.197} C_VEL
LIN {X 0,Y 206.898,Z 761.497,A -85,B 0,C 180,E1 -21046.245,E2 -21046.245} C_VEL
LIN {X 0,Y 207.104,Z 761.485,A -85,B 0,C 180,E1 -21050.231,E2 -21050.231} C_VEL
LIN {X 0,Y 207.071,Z 761.496,A -85,B 0,C 180,E1 -21054.156,E2 -21054.156} C_VEL
LIN {X 0,Y 207.384,Z 761.424,A -85,B 0,C 180,E1 -21058.058,E2 -21058.058} C_VEL
LIN {X 0,Y 207.517,Z 761.429,A -85,B 0,C 180,E1 -21060,E2 -21060} C_VEL
LIN {X 0,Y 207.387,Z 761.462,A -85,B 0,C 180,E1 -21061.942,E2 -21061.942} C_VEL
LIN {X 0,Y 207.17,Z 761.451,A -85,B 0,C 180,E1 -21067.799,E2 -21067.799} C_VEL
LIN {X 0,Y 206.941,Z 761.518,A -85,B 0,C 180,E1 -21071.758,E2 -21071.758} C_VEL
LIN {X 0,Y 206.835,Z 761.507,A -85,B 0,C 180,E1 -21075.773,E2 -21075.773} C_VEL
LIN {X 0,Y 206.752,Z 761.533,A -85,B 0,C 180,E1 -21079.873,E2 -21079.873} C_VEL
LIN {X 0,Y 206.748,Z 761.526,A -85,B 0,C 180,E1 -21084.074,E2 -21084.074} C_VEL
LIN {X 0,Y 206.738,Z 761.539,A -85,B 0,C 180,E1 -21088.42,E2 -21088.42} C_VEL
LIN {X 0,Y 206.7,Z 761.528,A -85,B 0,C 180,E1 -21092.958,E2 -21092.958} C_VEL
LIN {X 0,Y 206.682,Z 761.549,A -85,B 0,C 180,E1 -21097.74,E2 -21097.74} C_VEL
LIN {X 0,Y 206.64,Z 761.492,A -85,B 0,C 180,E1 -21101.562,E2 -21101.562} C_VEL
LIN {X 0,Y 206.633,Z 761.525,A -85,B 0,C 180,E1 -21105.582,E2 -21105.582} C_VEL
LIN {X 0,Y 206.662,Z 761.529,A -85,B 0,C 180,E1 -21109.749,E2 -21109.749} C_VEL
LIN {X 0,Y 206.7,Z 761.547,A -85,B 0,C 180,E1 -21114.689,E2 -21114.689} C_VEL
LIN {X 0,Y 206.75,Z 761.694,A -85,B 0,C 180,E1 -21118.296,E2 -21118.296} C_VEL
LIN {X 0,Y 207.007,Z 762.779,A -85,B 0,C 180,E1 -21118.685,E2 -21118.685} C_VEL
LIN {X 0,Y 212.335,Z 772.982,A -85,B 0,C 180,E1 -21119.977,E2 -21119.977} C_VEL
LIN {X 0,Y 218.012,Z 786.333,A -85,B 0,C 180,E1 -21121.337,E2 -21121.337} C_VEL
LIN {X 0,Y 221.109,Z 795.024,A -85,B 0,C 180,E1 -21122.093,E2 -21122.093} C_VEL
LIN {X 0,Y 221.322,Z 798.846,A -85,B 0,C 180,E1 -21122.26,E2 -21122.26} C_VEL
LIN {X 0,Y 219.948,Z 836.678,A -85,B 0,C 180,E1 -21123.497,E2 -21123.497} C_VEL
LIN {X 0,Y 219.43,Z 845.282,A -85,B 0,C 180,E1 -21123.99,E2 -21123.99} C_VEL
LIN {X 0,Y 218.477,Z 854.235,A -85,B 0,C 180,E1 -21124.705,E2 -21124.705} C_VEL
LIN {X 0,Y 217.179,Z 862.961,A -85,B 0,C 180,E1 -21125.632,E2 -21125.632} C_VEL
LIN {X 0,Y 215.761,Z 872.502,A -85,B 0,C 180,E1 -21126.991,E2 -21126.991} C_VEL
LIN {X 0,Y 213.684,Z 882.25,A -85,B 0,C 180,E1 -21128.79,E2 -21128.79} C_VEL
LIN {X 0,Y 211.923,Z 889.96,A -85,B 0,C 180,E1 -21130.632,E2 -21130.632} C_VEL
LIN {X 0,Y 210.367,Z 896.295,A -85,B 0,C 180,E1 -21132.502,E2 -21132.502} C_VEL
LIN {X 0,Y 208.968,Z 901.56,A -85,B 0,C 180,E1 -21134.392,E2 -21134.392} C_VEL
LIN {X 0,Y 207.762,Z 905.955,A -85,B 0,C 180,E1 -21136.303,E2 -21136.303} C_VEL
LIN {X 0,Y 206.388,Z 911.12,A -85,B 0,C 180,E1 -21139.205,E2 -21139.205} C_VEL
LIN {X 0,Y 205.706,Z 913.767,A -85,B 0,C 180,E1 -21141.156,E2 -21141.156} C_VEL
LIN {X 0,Y 204.969,Z 916.666,A -85,B 0,C 180,E1 -21144.096,E2 -21144.096} C_VEL
LIN {X 0,Y 204.676,Z 917.928,A -85,B 0,C 180,E1 -21146.062,E2 -21146.062} C_VEL
LIN {X 0,Y 204.526,Z 918.722,A -85,B 0,C 180,E1 -21148.031,E2 -21148.031} C_VEL
LIN {X 0,Y 204.5,Z 919.024,A -85,B 0,C 180,E1 -21150,E2 -21150} C_VEL
LIN {X 0,Y 204.524,Z 918.745,A -85,B 0,C 180,E1 -21151.969,E2 -21151.969} C_VEL
LIN {X 0,Y 204.672,Z 917.996,A -85,B 0,C 180,E1 -21153.938,E2 -21153.938} C_VEL
LIN {X 0,Y 205.03,Z 916.499,A -85,B 0,C 180,E1 -21156.246,E2 -21156.246} C_VEL
LIN {X 0,Y 205.643,Z 913.929,A -85,B 0,C 180,E1 -21158.847,E2 -21158.847} C_VEL
LIN {X 0,Y 206.329,Z 911.332,A -85,B 0,C 180,E1 -21160.798,E2 -21160.798} C_VEL
LIN {X 0,Y 207.696,Z 906.224,A -85,B 0,C 180,E1 -21163.702,E2 -21163.702} C_VEL
LIN {X 0,Y 209.247,Z 900.723,A -85,B 0,C 180,E1 -21166.087,E2 -21166.087} C_VEL
LIN {X 0,Y 211.12,Z 893.804,A -85,B 0,C 180,E1 -21168.436,E2 -21168.436} C_VEL
LIN {X 0,Y 212.921,Z 885.863,A -85,B 0,C 180,E1 -21170.53,E2 -21170.53} C_VEL
LIN {X 0,Y 214.595,Z 878.285,A -85,B 0,C 180,E1 -21172.125,E2 -21172.125} C_VEL
LIN {X 0,Y 216.174,Z 870.335,A -85,B 0,C 180,E1 -21173.469,E2 -21173.469} C_VEL
LIN {X 0,Y 217.51,Z 862.118,A -85,B 0,C 180,E1 -21174.583,E2 -21174.583} C_VEL
LIN {X 0,Y 218.594,Z 854.31,A -85,B 0,C 180,E1 -21175.412,E2 -21175.412} C_VEL
LIN {X 0,Y 219.457,Z 844.91,A -85,B 0,C 180,E1 -21176.176,E2 -21176.176} C_VEL
LIN {X 0,Y 220.052,Z 835.918,A -85,B 0,C 180,E1 -21176.668,E2 -21176.668} C_VEL
LIN {X 0,Y 221.342,Z 796.039,A -85,B 0,C 180,E1 -21177.98,E2 -21177.98} C_VEL
LIN {X 0,Y 219.214,Z 789.273,A -85,B 0,C 180,E1 -21178.526,E2 -21178.526} C_VEL
LIN {X 0,Y 212.983,Z 774.242,A -85,B 0,C 180,E1 -21180.02,E2 -21180.02} C_VEL
LIN {X 0,Y 208.213,Z 765.04,A -85,B 0,C 180,E1 -21181.151,E2 -21181.151} C_VEL
LIN {X 0,Y 206.924,Z 762.5,A -85,B 0,C 180,E1 -21181.521,E2 -21181.521} C_VEL
LIN {X 0,Y 206.728,Z 761.606,A -85,B 0,C 180,E1 -21181.948,E2 -21181.948} C_VEL
LIN {X 0,Y 206.7,Z 761.551,A -85,B 0,C 180,E1 -21185.311,E2 -21185.311} C_VEL
LIN {X 0,Y 206.662,Z 761.527,A -85,B 0,C 180,E1 -21190.251,E2 -21190.251} C_VEL
LIN {X 0,Y 206.633,Z 761.529,A -85,B 0,C 180,E1 -21194.418,E2 -21194.418} C_VEL
LIN {X 0,Y 206.64,Z 761.491,A -85,B 0,C 180,E1 -21198.438,E2 -21198.438} C_VEL
LIN {X 0,Y 206.682,Z 761.549,A -85,B 0,C 180,E1 -21202.26,E2 -21202.26} C_VEL
LIN {X 0,Y 206.7,Z 761.528,A -85,B 0,C 180,E1 -21207.042,E2 -21207.042} C_VEL
LIN {X 0,Y 206.766,Z 761.529,A -85,B 0,C 180,E1 -21212.098,E2 -21212.098} C_VEL
LIN {X 0,Y 206.756,Z 761.534,A -85,B 0,C 180,E1 -21216.604,E2 -21216.604} C_VEL
LIN {X 0,Y 206.869,Z 761.496,A -85,B 0,C 180,E1 -21222.196,E2 -21222.196} C_VEL
LIN {X 0,Y 206.885,Z 761.524,A -85,B 0,C 180,E1 -21226.243,E2 -21226.243} C_VEL
LIN {X 0,Y 207.134,Z 761.475,A -85,B 0,C 180,E1 -21230.232,E2 -21230.232} C_VEL
LIN {X 0,Y 207.077,Z 761.474,A -85,B 0,C 180,E1 -21234.156,E2 -21234.156} C_VEL
LIN {X 0,Y 207.387,Z 761.462,A -85,B 0,C 180,E1 -21238.058,E2 -21238.058} C_VEL
LIN {X 0,Y 207.517,Z 761.43,A -85,B 0,C 180,E1 -21240,E2 -21240} C_VEL
LIN {X 0,Y 207.383,Z 761.425,A -85,B 0,C 180,E1 -21241.942,E2 -21241.942} C_VEL
LIN {X 0,Y 207.165,Z 761.492,A -85,B 0,C 180,E1 -21247.799,E2 -21247.799} C_VEL
LIN {X 0,Y 206.945,Z 761.483,A -85,B 0,C 180,E1 -21251.757,E2 -21251.757} C_VEL
LIN {X 0,Y 206.869,Z 761.524,A -85,B 0,C 180,E1 -21255.77,E2 -21255.77} C_VEL
LIN {X 0,Y 206.785,Z 761.515,A -85,B 0,C 180,E1 -21259.869,E2 -21259.869} C_VEL
LIN {X 0,Y 206.765,Z 761.534,A -85,B 0,C 180,E1 -21264.072,E2 -21264.072} C_VEL
LIN {X 0,Y 206.738,Z 761.523,A -85,B 0,C 180,E1 -21268.419,E2 -21268.419} C_VEL
LIN {X 0,Y 206.707,Z 761.55,A -85,B 0,C 180,E1 -21272.956,E2 -21272.956} C_VEL
